C07316=1207.286,250.336,-62.631,-177.060,6.729,148.376
C07317=1207.282,250.584,-62.658,-177.057,6.731,148.376
C07318=1207.277,250.833,-62.684,-177.054,6.733,148.376
C07319=1207.273,251.081,-62.711,-177.052,6.736,148.376
C07320=1207.269,251.330,-62.737,-177.049,6.737,148.375
C07321=1207.264,251.578,-62.764,-177.047,6.740,148.375
C07322=1207.259,251.827,-62.791,-177.044,6.742,148.375
C07323=1207.255,252.075,-62.817,-177.042,6.744,148.375
C07324=1207.251,252.325,-62.844,-177.039,6.746,148.375
C07325=1207.247,252.573,-62.871,-177.037,6.749,148.375
C07326=1207.243,252.821,-62.898,-177.034,6.751,148.374
C07327=1207.238,253.070,-62.925,-177.031,6.753,148.374
C07328=1207.233,253.318,-62.952,-177.029,6.756,148.374
C07329=1207.229,253.566,-62.978,-177.026,6.758,148.374
C07330=1207.224,253.815,-63.005,-177.024,6.760,148.374
C07331=1207.220,254.064,-63.032,-177.021,6.762,148.373
C07332=1207.215,254.312,-63.059,-177.018,6.765,148.373
C07333=1207.211,254.561,-63.085,-177.016,6.767,148.373
C07334=1207.207,254.809,-63.112,-177.014,6.769,148.373
C07335=1207.202,255.058,-63.140,-177.011,6.771,148.372
C07336=1207.197,255.306,-63.167,-177.008,6.774,148.372
C07337=1207.194,255.555,-63.193,-177.006,6.776,148.372
C07338=1207.189,255.804,-63.220,-177.004,6.778,148.372
C07339=1207.185,256.052,-63.248,-177.000,6.781,148.372
C07340=1207.180,256.301,-63.275,-176.998,6.783,148.372
C07341=1207.176,256.549,-63.301,-176.996,6.785,148.371
C07342=1207.171,256.797,-63.328,-176.994,6.787,148.371
C07343=1207.167,257.046,-63.355,-176.990,6.789,148.371
C07344=1207.162,257.294,-63.382,-176.988,6.792,148.371
C07345=1207.157,257.543,-63.409,-176.986,6.793,148.371
C07346=1207.153,257.792,-63.437,-176.983,6.797,148.371
C07347=1207.150,258.039,-63.464,-176.980,6.798,148.370
C07348=1207.145,258.288,-63.491,-176.978,6.801,148.370
C07349=1207.140,258.536,-63.518,-176.975,6.803,148.370
C07350=1207.136,258.785,-63.545,-176.973,6.805,148.370
C07351=1207.131,259.033,-63.572,-176.970,6.807,148.370
C07352=1207.127,259.283,-63.600,-176.968,6.809,148.369
C07353=1207.122,259.531,-63.627,-176.965,6.812,148.369
C07354=1207.118,259.779,-63.654,-176.963,6.814,148.369
C07355=1207.114,260.027,-63.681,-176.960,6.816,148.369
C07356=1207.109,260.276,-63.708,-176.957,6.819,148.369
C07357=1207.105,260.525,-63.735,-176.955,6.821,148.368
C07358=1207.101,260.773,-63.762,-176.953,6.823,148.368
C07359=1207.096,261.021,-63.790,-176.949,6.826,148.368
C07360=1207.092,261.270,-63.817,-176.947,6.828,148.368
C07361=1207.087,261.518,-63.844,-176.945,6.830,148.368
C07362=1207.083,261.767,-63.872,-176.942,6.833,148.368
C07363=1207.079,262.015,-63.900,-176.939,6.835,148.367
C07364=1207.074,262.264,-63.927,-176.937,6.837,148.367
C07365=1207.069,262.512,-63.954,-176.934,6.840,148.367
C07366=1207.065,262.785,-63.984,-176.932,6.842,148.367
C07367=1207.060,263.058,-64.014,-176.929,6.845,148.367
C07368=1207.055,263.331,-64.044,-176.926,6.848,148.367
C07369=1207.050,263.603,-64.074,-176.923,6.850,148.366
C07370=1207.046,263.852,-64.102,-176.921,6.853,148.366
C07371=1207.042,264.100,-64.129,-176.918,6.854,148.366
C07372=1207.037,264.348,-64.156,-176.916,6.857,148.366
C07373=1207.033,264.597,-64.183,-176.913,6.859,148.366
C07374=1207.029,264.846,-64.212,-176.911,6.861,148.366
C07375=1207.024,265.094,-64.239,-176.908,6.863,148.365
C07376=1207.019,265.342,-64.267,-176.905,6.866,148.365
C07377=1207.015,265.591,-64.294,-176.903,6.868,148.365
C07378=1207.011,265.839,-64.322,-176.901,6.870,148.365
C07379=1207.006,266.088,-64.349,-176.898,6.873,148.365
C07380=1207.002,266.336,-64.377,-176.895,6.875,148.365
C07381=1206.998,266.585,-64.404,-176.893,6.877,148.364
C07382=1206.993,266.833,-64.432,-176.890,6.880,148.364
C07383=1206.989,267.081,-64.459,-176.888,6.882,148.364
C07384=1206.985,267.330,-64.487,-176.886,6.885,148.364
C07385=1206.980,267.579,-64.515,-176.883,6.887,148.364
C07386=1206.975,267.826,-64.543,-176.880,6.889,148.364
C07387=1206.971,268.076,-64.570,-176.877,6.892,148.363
C07388=1206.967,268.324,-64.598,-176.875,6.894,148.363
C07389=1206.962,268.571,-64.626,-176.873,6.896,148.363
C07390=1206.958,268.821,-64.653,-176.870,6.899,148.363
C07391=1206.953,269.069,-64.682,-176.868,6.901,148.363
C07392=1206.949,269.317,-64.709,-176.865,6.903,148.363
C07393=1206.945,269.566,-64.737,-176.862,6.906,148.363
C07394=1206.941,269.814,-64.765,-176.860,6.908,148.363
C07395=1206.936,270.063,-64.792,-176.857,6.911,148.362
C07396=1206.931,270.311,-64.820,-176.855,6.913,148.362
C07397=1206.927,270.559,-64.848,-176.852,6.915,148.362
C07398=1206.923,270.808,-64.876,-176.850,6.918,148.362
C07399=1206.919,271.056,-64.903,-176.847,6.920,148.362
C07400=1206.914,271.304,-64.932,-176.845,6.922,148.361
C07401=1206.910,271.553,-64.960,-176.842,6.925,148.361
C07402=1206.905,271.801,-64.987,-176.840,6.927,148.361
C07403=1206.901,272.050,-65.015,-176.837,6.930,148.361
C07404=1206.896,272.298,-65.044,-176.835,6.932,148.361
C07405=1206.893,272.547,-65.072,-176.832,6.934,148.361
C07406=1206.888,272.795,-65.099,-176.829,6.937,148.361
C07407=1206.883,273.043,-65.127,-176.827,6.939,148.361
C07408=1206.879,273.292,-65.155,-176.824,6.942,148.360
C07409=1206.875,273.540,-65.183,-176.822,6.944,148.360
C07410=1206.870,273.789,-65.212,-176.820,6.946,148.360
C07411=1206.866,274.037,-65.240,-176.817,6.949,148.360
C07412=1206.862,274.285,-65.268,-176.814,6.951,148.360
C07413=1206.857,274.533,-65.296,-176.812,6.954,148.360
C07414=1206.853,274.783,-65.323,-176.809,6.956,148.360
C07415=1206.849,275.030,-65.351,-176.806,6.959,148.360
C07416=1206.844,275.279,-65.380,-176.804,6.961,148.359
C07417=1206.840,275.527,-65.408,-176.802,6.963,148.359
C07418=1206.835,275.775,-65.436,-176.799,6.966,148.359
C07419=1206.831,276.024,-65.464,-176.797,6.969,148.359
C07420=1206.827,276.272,-65.492,-176.794,6.971,148.359
C07421=1206.822,276.521,-65.521,-176.792,6.973,148.359
C07422=1206.818,276.769,-65.549,-176.789,6.976,148.359
C07423=1206.813,277.017,-65.577,-176.786,6.978,148.358
C07424=1206.810,277.266,-65.605,-176.784,6.980,148.358
C07425=1206.805,277.514,-65.633,-176.781,6.984,148.358
C07426=1206.801,277.763,-65.662,-176.779,6.985,148.358
C07427=1206.796,278.011,-65.690,-176.776,6.988,148.358
C07428=1206.792,278.260,-65.718,-176.774,6.991,148.358
C07429=1206.787,278.507,-65.746,-176.771,6.994,148.358
C07430=1206.783,278.756,-65.775,-176.769,6.995,148.358
C07431=1206.779,279.004,-65.803,-176.767,6.998,148.357
C07432=1206.774,279.252,-65.832,-176.764,7.001,148.357
C07433=1206.770,279.500,-65.860,-176.761,7.003,148.357
C07434=1206.766,279.749,-65.889,-176.759,7.006,148.357
C07435=1206.762,279.998,-65.917,-176.756,7.008,148.357
C07436=1206.757,280.246,-65.945,-176.754,7.011,148.357
C07437=1206.753,280.495,-65.973,-176.751,7.013,148.357
C07438=1206.748,280.742,-66.002,-176.748,7.016,148.357
C07439=1206.744,280.991,-66.031,-176.746,7.018,148.357
C07440=1206.739,281.239,-66.059,-176.744,7.020,148.356
C07441=1206.735,281.488,-66.088,-176.741,7.023,148.356
C07442=1206.731,281.736,-66.117,-176.739,7.025,148.356
C07443=1206.726,281.984,-66.145,-176.736,7.028,148.356
C07444=1206.723,282.232,-66.173,-176.734,7.030,148.356
C07445=1206.718,282.481,-66.201,-176.731,7.033,148.356
C07446=1206.713,282.729,-66.231,-176.729,7.035,148.356
C07447=1206.710,282.978,-66.259,-176.726,7.038,148.356
C07448=1206.705,283.226,-66.287,-176.723,7.040,148.356
C07449=1206.700,283.475,-66.316,-176.721,7.043,148.355
C07450=1206.697,283.723,-66.345,-176.719,7.045,148.355
C07451=1206.692,283.971,-66.373,-176.716,7.048,148.355
C07452=1206.687,284.220,-66.402,-176.713,7.050,148.355
C07453=1206.684,284.468,-66.431,-176.711,7.052,148.355
C07454=1206.679,284.716,-66.459,-176.708,7.055,148.355
C07455=1206.674,284.964,-66.489,-176.706,7.057,148.355
C07456=1206.671,285.213,-66.517,-176.704,7.060,148.355
C07457=1206.665,285.461,-66.545,-176.701,7.062,148.355
C07458=1206.661,285.709,-66.575,-176.698,7.065,148.355
C07459=1206.658,285.958,-66.603,-176.696,7.068,148.355
C07460=1206.653,286.205,-66.632,-176.694,7.071,148.354
C07461=1206.648,286.454,-66.661,-176.691,7.072,148.354
C07462=1206.644,286.702,-66.690,-176.688,7.076,148.354
C07463=1206.640,286.950,-66.718,-176.686,7.078,148.354
C07464=1206.636,287.199,-66.747,-176.683,7.081,148.354
C07465=1206.631,287.447,-66.776,-176.681,7.083,148.354
C07466=1206.626,287.695,-66.805,-176.678,7.086,148.354
C07467=1206.623,287.944,-66.833,-176.676,7.088,148.354
C07468=1206.618,288.192,-66.863,-176.673,7.091,148.354
C07469=1206.614,288.441,-66.892,-176.671,7.093,148.354
C07470=1206.609,288.714,-66.924,-176.668,7.096,148.354
C07471=1206.605,288.989,-66.956,-176.665,7.099,148.353
C07472=1206.599,289.263,-66.988,-176.663,7.102,148.353
C07473=1206.595,289.537,-67.020,-176.660,7.105,148.353
C07474=1206.590,289.786,-67.049,-176.658,7.107,148.353
C07475=1206.586,290.033,-67.077,-176.655,7.110,148.353
C07476=1206.582,290.282,-67.106,-176.653,7.112,148.353
C07477=1206.577,290.531,-67.136,-176.650,7.115,148.353
C07478=1206.573,290.779,-67.165,-176.648,7.117,148.353
C07479=1206.569,291.028,-67.194,-176.645,7.120,148.353
C07480=1206.564,291.275,-67.223,-176.643,7.122,148.353
C07481=1206.560,291.523,-67.252,-176.640,7.125,148.353
C07482=1206.556,291.772,-67.282,-176.638,7.127,148.352
C07483=1206.552,292.020,-67.310,-176.635,7.130,148.352
C07484=1206.548,292.269,-67.339,-176.633,7.132,148.352
C07485=1206.543,292.516,-67.369,-176.630,7.135,148.352
C07486=1206.539,292.764,-67.398,-176.628,7.138,148.352
C07487=1206.534,293.013,-67.427,-176.625,7.141,148.352
C07488=1206.530,293.262,-67.456,-176.623,7.143,148.352
C07489=1206.526,293.510,-67.486,-176.620,7.146,148.352
C07490=1206.521,293.757,-67.515,-176.618,7.148,148.352
C07491=1206.517,294.006,-67.544,-176.615,7.151,148.352
C07492=1206.513,294.254,-67.574,-176.612,7.154,148.352
C07493=1206.508,294.503,-67.602,-176.610,7.156,148.352
C07494=1206.504,294.751,-67.632,-176.608,7.159,148.352
C07495=1206.500,294.999,-67.661,-176.605,7.161,148.352
C07496=1206.496,295.248,-67.691,-176.603,7.164,148.352
C07497=1206.491,295.495,-67.720,-176.601,7.166,148.352
C07498=1206.487,295.743,-67.749,-176.598,7.169,148.352
C07499=1206.482,295.992,-67.779,-176.595,7.171,148.351
C07500=1206.478,296.240,-67.808,-176.593,7.174,148.351
C07501=1206.474,296.488,-67.838,-176.591,7.177,148.351
C07502=1206.470,296.737,-67.867,-176.588,7.180,148.351
C07503=1206.466,296.985,-67.897,-176.586,7.182,148.351
C07504=1206.462,297.233,-67.926,-176.583,7.185,148.351
C07505=1206.457,297.481,-67.955,-176.580,7.188,148.351
C07506=1206.453,297.729,-67.984,-176.578,7.190,148.351
C07507=1206.448,297.978,-68.015,-176.576,7.193,148.351
C07508=1206.443,298.226,-68.044,-176.573,7.195,148.351
C07509=1206.439,298.474,-68.073,-176.571,7.198,148.351
C07510=1206.435,298.722,-68.103,-176.569,7.201,148.351
C07511=1206.431,298.971,-68.132,-176.566,7.204,148.351
C07512=1206.427,299.219,-68.162,-176.564,7.206,148.351
C07513=1206.423,299.467,-68.191,-176.561,7.209,148.351
C07514=1206.418,299.715,-68.221,-176.559,7.211,148.351
C07515=1206.413,299.964,-68.251,-176.556,7.214,148.351
C07516=1206.409,300.212,-68.280,-176.554,7.217,148.351
C07517=1206.405,300.460,-68.310,-176.551,7.219,148.351
C07518=1206.401,300.708,-68.340,-176.549,7.222,148.351
C07519=1206.397,300.956,-68.369,-176.547,7.224,148.351
C07520=1206.392,301.205,-68.399,-176.544,7.227,148.351
C07521=1206.388,301.453,-68.429,-176.542,7.230,148.351
C07522=1206.384,301.701,-68.459,-176.539,7.233,148.350
C07523=1206.380,301.949,-68.488,-176.536,7.236,148.350
C07524=1206.376,302.197,-68.518,-176.534,7.238,148.350
C07525=1206.371,302.446,-68.548,-176.532,7.241,148.350
C07526=1206.367,302.694,-68.578,-176.530,7.243,148.350
C07527=1206.363,302.942,-68.608,-176.527,7.246,148.350
C07528=1206.359,303.190,-68.637,-176.525,7.248,148.350
C07529=1206.354,303.439,-68.667,-176.522,7.251,148.350
C07530=1206.350,303.686,-68.697,-176.519,7.254,148.350
C07531=1206.346,303.935,-68.727,-176.517,7.257,148.350
C07532=1206.341,304.183,-68.757,-176.515,7.260,148.350
C07533=1206.337,304.431,-68.787,-176.512,7.262,148.350
C07534=1206.333,304.679,-68.816,-176.510,7.265,148.350
C07535=1206.328,304.928,-68.846,-176.508,7.267,148.350
C07536=1206.324,305.175,-68.877,-176.505,7.270,148.350
C07537=1206.320,305.424,-68.906,-176.502,7.273,148.350
C07538=1206.315,305.672,-68.937,-176.500,7.275,148.350
C07539=1206.311,305.920,-68.966,-176.497,7.278,148.350
C07540=1206.307,306.168,-68.996,-176.495,7.281,148.350
C07541=1206.302,306.416,-69.026,-176.493,7.284,148.350
C07542=1206.298,306.664,-69.056,-176.490,7.286,148.350
C07543=1206.294,306.912,-69.086,-176.488,7.289,148.350
C07544=1206.289,307.161,-69.116,-176.485,7.292,148.350
C07545=1206.285,307.408,-69.146,-176.483,7.294,148.350
C07546=1206.280,307.657,-69.176,-176.481,7.297,148.350
C07547=1206.277,307.905,-69.207,-176.479,7.300,148.350
C07548=1206.272,308.154,-69.237,-176.476,7.303,148.350
C07549=1206.268,308.401,-69.267,-176.473,7.306,148.350
C07550=1206.264,308.650,-69.297,-176.471,7.308,148.350
C07551=1206.259,308.898,-69.327,-176.468,7.311,148.350
C07552=1206.256,309.145,-69.357,-176.466,7.313,148.350
C07553=1206.251,309.394,-69.388,-176.464,7.316,148.350
C07554=1206.247,309.642,-69.418,-176.461,7.319,148.350
C07555=1206.242,309.890,-69.448,-176.459,7.322,148.350
C07556=1206.239,310.138,-69.478,-176.457,7.325,148.350
C07557=1206.234,310.386,-69.509,-176.454,7.327,148.350
C07558=1206.230,310.635,-69.538,-176.452,7.330,148.350
C07559=1206.225,310.883,-69.569,-176.449,7.333,148.350
C07560=1206.221,311.130,-69.599,-176.447,7.335,148.350
C07561=1206.216,311.379,-69.629,-176.445,7.338,148.350
C07562=1206.213,311.627,-69.660,-176.443,7.341,148.350
C07563=1206.208,311.875,-69.691,-176.440,7.344,148.350
C07564=1206.204,312.123,-69.720,-176.437,7.347,148.350
C07565=1206.200,312.371,-69.751,-176.435,7.349,148.350
C07566=1206.195,312.619,-69.782,-176.432,7.352,148.350
C07567=1206.191,312.867,-69.812,-176.431,7.354,148.350
C07568=1206.187,313.116,-69.842,-176.428,7.357,148.350
C07569=1206.183,313.364,-69.873,-176.425,7.360,148.350
C07570=1206.178,313.612,-69.903,-176.423,7.363,148.350
C07571=1206.174,313.860,-69.933,-176.421,7.366,148.350
C07572=1206.170,314.107,-69.964,-176.419,7.368,148.350
C07573=1206.166,314.357,-69.995,-176.416,7.371,148.350
C07574=1206.161,314.633,-70.029,-176.414,7.374,148.350
C07575=1206.157,314.908,-70.063,-176.411,7.377,148.350
C07576=1206.152,315.184,-70.096,-176.408,7.380,148.350
C07577=1206.147,315.460,-70.130,-176.406,7.383,148.350
C07578=1206.143,315.709,-70.162,-176.403,7.387,148.350
C07579=1206.138,315.957,-70.192,-176.401,7.389,148.350
C07580=1206.134,316.204,-70.222,-176.399,7.392,148.350
C07581=1206.129,316.453,-70.253,-176.396,7.395,148.350
C07582=1206.125,316.702,-70.284,-176.394,7.397,148.350
C07583=1206.122,316.949,-70.314,-176.392,7.401,148.350
C07584=1206.117,317.197,-70.345,-176.389,7.403,148.350
C07585=1206.113,317.446,-70.376,-176.387,7.406,148.350
C07586=1206.108,317.694,-70.406,-176.385,7.409,148.351
C07587=1206.104,317.942,-70.437,-176.382,7.411,148.350
C07588=1206.100,318.190,-70.467,-176.380,7.414,148.350
C07589=1206.096,318.438,-70.499,-176.377,7.418,148.351
C07590=1206.092,318.686,-70.529,-176.375,7.420,148.351
C07591=1206.088,318.933,-70.560,-176.373,7.423,148.351
C07592=1206.084,319.182,-70.591,-176.371,7.425,148.351
C07593=1206.079,319.430,-70.622,-176.368,7.428,148.351
C07594=1206.074,319.678,-70.653,-176.366,7.431,148.351
C07595=1206.071,319.926,-70.683,-176.364,7.434,148.351
C07596=1206.067,320.174,-70.714,-176.361,7.437,148.351
C07597=1206.062,320.422,-70.745,-176.359,7.440,148.351
C07598=1206.058,320.671,-70.776,-176.357,7.442,148.351
C07599=1206.053,320.919,-70.807,-176.354,7.446,148.351
C07600=1206.050,321.166,-70.838,-176.352,7.448,148.351
C07601=1206.046,321.414,-70.869,-176.349,7.451,148.351
C07602=1206.041,321.662,-70.900,-176.347,7.454,148.351
C07603=1206.036,321.910,-70.930,-176.345,7.456,148.351
C07604=1206.032,322.159,-70.961,-176.342,7.459,148.351
C07605=1206.028,322.406,-70.993,-176.340,7.463,148.351
C07606=1206.025,322.655,-71.023,-176.338,7.465,148.351
C07607=1206.020,322.903,-71.054,-176.336,7.468,148.352
C07608=1206.016,323.151,-71.085,-176.334,7.470,148.352
C07609=1206.012,323.399,-71.117,-176.331,7.474,148.352
C07610=1206.007,323.647,-71.148,-176.329,7.477,148.352
C07611=1206.003,323.895,-71.179,-176.327,7.479,148.352
C07612=1205.999,324.143,-71.210,-176.325,7.482,148.352
C07613=1205.994,324.390,-71.241,-176.322,7.485,148.352
C07614=1205.990,324.639,-71.272,-176.320,7.488,148.352
C07615=1205.986,324.886,-71.304,-176.318,7.491,148.352
C07616=1205.982,325.135,-71.335,-176.315,7.493,148.352
C07617=1205.977,325.383,-71.366,-176.313,7.497,148.352
C07618=1205.974,325.631,-71.397,-176.311,7.500,148.352
C07619=1205.970,325.879,-71.428,-176.309,7.502,148.352
C07620=1205.966,326.126,-71.459,-176.306,7.505,148.352
C07621=1205.962,326.375,-71.490,-176.304,7.508,148.352
C07622=1205.957,326.623,-71.521,-176.302,7.511,148.353
C07623=1205.953,326.871,-71.553,-176.299,7.514,148.353
C07624=1205.949,327.119,-71.584,-176.298,7.516,148.353
C07625=1205.944,327.367,-71.616,-176.295,7.519,148.353
C07626=1205.940,327.615,-71.647,-176.293,7.523,148.353
C07627=1205.936,327.863,-71.679,-176.290,7.525,148.353
C07628=1205.931,328.111,-71.709,-176.288,7.528,148.353
C07629=1205.928,328.359,-71.741,-176.286,7.531,148.353
C07630=1205.923,328.607,-71.772,-176.284,7.534,148.353
C07631=1205.919,328.855,-71.804,-176.281,7.537,148.353
C07632=1205.915,329.103,-71.835,-176.279,7.540,148.354
C07633=1205.911,329.351,-71.866,-176.277,7.542,148.354
C07634=1205.907,329.598,-71.898,-176.275,7.546,148.354
C07635=1205.903,329.847,-71.929,-176.273,7.548,148.354
C07636=1205.898,330.094,-71.960,-176.270,7.551,148.354
C07637=1205.894,330.343,-71.992,-176.268,7.554,148.354
C07638=1205.889,330.591,-72.024,-176.266,7.557,148.354
C07639=1205.885,330.839,-72.056,-176.264,7.560,148.354
C07640=1205.881,331.087,-72.086,-176.261,7.563,148.354
C07641=1205.877,331.335,-72.118,-176.259,7.566,148.354
C07642=1205.873,331.582,-72.150,-176.257,7.569,148.354
C07643=1205.869,331.831,-72.181,-176.255,7.571,148.355
C07644=1205.865,332.078,-72.212,-176.253,7.574,148.355
C07645=1205.860,332.326,-72.245,-176.250,7.577,148.355
C07646=1205.856,332.575,-72.276,-176.249,7.580,148.355
C07647=1205.852,332.822,-72.307,-176.246,7.583,148.355
C07648=1205.848,333.070,-72.339,-176.244,7.586,148.355
C07649=1205.844,333.318,-72.371,-176.242,7.589,148.355
C07650=1205.839,333.566,-72.403,-176.239,7.592,148.355
C07651=1205.835,333.814,-72.434,-176.237,7.595,148.356
C07652=1205.831,334.062,-72.466,-176.235,7.598,148.356
C07653=1205.827,334.310,-72.497,-176.233,7.601,148.356
C07654=1205.822,334.558,-72.530,-176.231,7.603,148.356
C07655=1205.819,334.806,-72.561,-176.229,7.607,148.356
C07656=1205.814,335.054,-72.592,-176.226,7.610,148.356
C07657=1205.810,335.302,-72.624,-176.225,7.612,148.356
C07658=1205.806,335.550,-72.656,-176.222,7.616,148.357
C07659=1205.801,335.798,-72.688,-176.220,7.619,148.357
C07660=1205.798,336.046,-72.720,-176.218,7.621,148.357
C07661=1205.793,336.294,-72.752,-176.216,7.624,148.357
C07662=1205.789,336.541,-72.784,-176.214,7.627,148.357
C07663=1205.785,336.789,-72.816,-176.212,7.630,148.357
C07664=1205.780,337.037,-72.848,-176.209,7.633,148.357
C07665=1205.777,337.285,-72.879,-176.207,7.636,148.357
C07666=1205.773,337.534,-72.911,-176.205,7.639,148.358
C07667=1205.768,337.781,-72.943,-176.203,7.642,148.358
C07668=1205.764,338.029,-72.975,-176.201,7.645,148.358
C07669=1205.760,338.277,-73.006,-176.198,7.648,148.358
C07670=1205.755,338.525,-73.038,-176.197,7.650,148.358
C07671=1205.751,338.773,-73.070,-176.195,7.654,148.358
C07672=1205.748,339.020,-73.103,-176.192,7.657,148.359
C07673=1205.743,339.269,-73.135,-176.191,7.659,148.359
C07674=1205.739,339.516,-73.167,-176.188,7.662,148.359
C07675=1205.735,339.765,-73.199,-176.186,7.666,148.359
C07676=1205.731,340.013,-73.231,-176.184,7.668,148.359
C07677=1205.727,340.260,-73.263,-176.182,7.672,148.359
C07678=1205.722,340.538,-73.299,-176.180,7.675,148.360
C07679=1205.717,340.817,-73.335,-176.177,7.678,148.360
C07680=1205.712,341.095,-73.371,-176.175,7.681,148.360
C07681=1205.708,341.373,-73.407,-176.173,7.685,148.360
C07682=1205.704,341.621,-73.439,-176.170,7.688,148.360
C07683=1205.699,341.869,-73.471,-176.169,7.691,148.361
C07684=1205.695,342.117,-73.503,-176.166,7.694,148.361
C07685=1205.691,342.365,-73.535,-176.164,7.697,148.361
C07686=1205.687,342.613,-73.568,-176.162,7.699,148.361
C07687=1205.683,342.860,-73.600,-176.160,7.703,148.361
C07688=1205.678,343.109,-73.632,-176.158,7.705,148.361
C07689=1205.675,343.357,-73.664,-176.156,7.709,148.362
C07690=1205.670,343.604,-73.697,-176.154,7.712,148.362
C07691=1205.666,343.852,-73.729,-176.152,7.715,148.362
C07692=1205.662,344.100,-73.761,-176.150,7.718,148.362
C07693=1205.658,344.348,-73.793,-176.148,7.720,148.362
C07694=1205.654,344.596,-73.826,-176.146,7.724,148.363
C07695=1205.649,344.843,-73.858,-176.144,7.727,148.363
C07696=1205.645,345.091,-73.890,-176.142,7.730,148.363
C07697=1205.641,345.339,-73.923,-176.140,7.733,148.363
C07698=1205.637,345.587,-73.955,-176.137,7.736,148.363
C07699=1205.633,345.836,-73.987,-176.136,7.738,148.363
C07700=1205.628,346.083,-74.020,-176.133,7.742,148.364
C07701=1205.624,346.331,-74.052,-176.132,7.744,148.364
C07702=1205.620,346.578,-74.085,-176.130,7.748,148.364
C07703=1205.617,346.826,-74.117,-176.127,7.751,148.364
C07704=1205.612,347.075,-74.149,-176.126,7.754,148.364
C07705=1205.608,347.322,-74.183,-176.124,7.757,148.365
C07706=1205.604,347.570,-74.214,-176.122,7.760,148.365
C07707=1205.600,347.818,-74.247,-176.120,7.763,148.365
C07708=1205.595,348.066,-74.280,-176.118,7.766,148.365
C07709=1205.592,348.313,-74.312,-176.116,7.769,148.366
C07710=1205.587,348.562,-74.345,-176.114,7.772,148.366
C07711=1205.583,348.809,-74.378,-176.112,7.775,148.366
C07712=1205.579,349.057,-74.409,-176.110,7.778,148.366
C07713=1205.575,349.304,-74.442,-176.108,7.781,148.367
C07714=1205.570,349.553,-74.475,-176.106,7.784,148.367
C07715=1205.567,349.800,-74.507,-176.104,7.787,148.367
C07716=1205.562,350.049,-74.540,-176.102,7.790,148.367
C07717=1205.558,350.296,-74.573,-176.100,7.793,148.367
C07718=1205.554,350.545,-74.605,-176.098,7.797,148.368
C07719=1205.550,350.791,-74.638,-176.097,7.799,148.368
C07720=1205.545,351.040,-74.670,-176.095,7.803,148.368
C07721=1205.541,351.287,-74.703,-176.093,7.805,148.368
C07722=1205.537,351.535,-74.736,-176.091,7.808,148.369
C07723=1205.533,351.783,-74.768,-176.089,7.811,148.369
C07724=1205.529,352.031,-74.801,-176.087,7.815,148.369
C07725=1205.525,352.279,-74.835,-176.085,7.818,148.369
C07726=1205.521,352.527,-74.867,-176.083,7.820,148.370
C07727=1205.517,352.775,-74.900,-176.081,7.824,148.370
C07728=1205.513,353.022,-74.933,-176.079,7.826,148.370
C07729=1205.509,353.271,-74.965,-176.078,7.830,148.370
C07730=1205.505,353.518,-74.998,-176.076,7.832,148.371
C07731=1205.500,353.765,-75.031,-176.074,7.836,148.371
C07732=1205.496,354.013,-75.064,-176.072,7.839,148.371
C07733=1205.492,354.261,-75.096,-176.070,7.842,148.371
C07734=1205.488,354.509,-75.129,-176.068,7.845,148.372
C07735=1205.484,354.756,-75.162,-176.067,7.848,148.372
C07736=1205.480,355.004,-75.196,-176.064,7.851,148.372
C07737=1205.475,355.253,-75.228,-176.063,7.854,148.372
C07738=1205.471,355.500,-75.261,-176.061,7.857,148.373
C07739=1205.467,355.748,-75.294,-176.059,7.861,148.373
C07740=1205.463,355.995,-75.327,-176.057,7.863,148.373
C07741=1205.459,356.243,-75.360,-176.055,7.867,148.374
C07742=1205.455,356.492,-75.392,-176.054,7.869,148.374
C07743=1205.451,356.739,-75.426,-176.052,7.873,148.374
C07744=1205.447,356.987,-75.459,-176.050,7.875,148.374
C07745=1205.442,357.235,-75.492,-176.048,7.879,148.375
C07746=1205.438,357.482,-75.525,-176.046,7.882,148.375
C07747=1205.434,357.730,-75.558,-176.045,7.885,148.375
C07748=1205.430,357.978,-75.591,-176.043,7.889,148.376
C07749=1205.426,358.226,-75.625,-176.041,7.891,148.376
C07750=1205.422,358.473,-75.658,-176.039,7.894,148.376
C07751=1205.418,358.721,-75.691,-176.038,7.897,148.376
C07752=1205.413,358.969,-75.724,-176.035,7.901,148.377
C07753=1205.409,359.217,-75.757,-176.034,7.903,148.377
C07754=1205.405,359.464,-75.790,-176.032,7.907,148.377
C07755=1205.401,359.712,-75.824,-176.031,7.910,148.378
C07756=1205.397,359.960,-75.857,-176.029,7.913,148.378
C07757=1205.393,360.207,-75.890,-176.027,7.916,148.378
C07758=1205.389,360.455,-75.923,-176.025,7.919,148.379
C07759=1205.385,360.704,-75.956,-176.024,7.922,148.379
C07760=1205.381,360.951,-75.990,-176.022,7.925,148.379
C07761=1205.377,361.199,-76.023,-176.021,7.928,148.380
C07762=1205.373,361.447,-76.056,-176.018,7.931,148.380
C07763=1205.369,361.695,-76.089,-176.017,7.934,148.380
C07764=1205.364,361.942,-76.122,-176.015,7.938,148.380
C07765=1205.360,362.190,-76.155,-176.014,7.940,148.381
C07766=1205.356,362.438,-76.189,-176.012,7.944,148.381
C07767=1205.352,362.685,-76.222,-176.010,7.947,148.381
C07768=1205.348,362.933,-76.255,-176.009,7.950,148.382
C07769=1205.344,363.180,-76.289,-176.007,7.953,148.382
C07770=1205.340,363.428,-76.322,-176.005,7.956,148.382
C07771=1205.336,363.676,-76.355,-176.004,7.959,148.383
C07772=1205.332,363.924,-76.389,-176.002,7.962,148.383
C07773=1205.328,364.172,-76.422,-176.001,7.965,148.383
C07774=1205.324,364.420,-76.455,-175.999,7.969,148.384
C07775=1205.319,364.667,-76.489,-175.997,7.971,148.384
C07776=1205.315,364.915,-76.523,-175.996,7.974,148.384
C07777=1205.311,365.163,-76.556,-175.994,7.978,148.385
C07778=1205.307,365.410,-76.589,-175.993,7.981,148.385
C07779=1205.304,365.658,-76.623,-175.991,7.984,148.386
C07780=1205.300,365.906,-76.656,-175.989,7.987,148.386
C07781=1205.295,366.154,-76.689,-175.988,7.990,148.386
C07782=1205.291,366.434,-76.728,-175.987,7.993,148.387
C07783=1205.285,366.714,-76.766,-175.985,7.997,148.387
C07784=1205.281,366.995,-76.803,-175.983,8.001,148.388
C07785=1205.276,367.276,-76.842,-175.981,8.004,148.388
C07786=1205.272,367.523,-76.875,-175.980,8.007,148.388
C07787=1205.268,367.770,-76.909,-175.978,8.010,148.389
C07788=1205.265,368.019,-76.942,-175.977,8.013,148.389
C07789=1205.261,368.267,-76.975,-175.975,8.016,148.390
C07790=1205.256,368.514,-77.010,-175.974,8.020,148.390
C07791=1205.252,368.762,-77.043,-175.972,8.022,148.390
C07792=1205.248,369.009,-77.077,-175.971,8.025,148.391
C07793=1205.244,369.257,-77.110,-175.969,8.029,148.391
C07794=1205.240,369.505,-77.144,-175.968,8.031,148.391
C07795=1205.236,369.752,-77.178,-175.967,8.034,148.392
C07796=1205.232,370.000,-77.211,-175.965,8.038,148.392
C07797=1205.228,370.247,-77.245,-175.964,8.041,148.393
C07798=1205.223,370.495,-77.279,-175.962,8.043,148.393
C07799=1205.220,370.743,-77.313,-175.961,8.047,148.393
C07800=1205.216,370.991,-77.346,-175.959,8.050,148.394
C07801=1205.211,371.238,-77.381,-175.958,8.053,148.394
C07802=1205.207,371.486,-77.414,-175.957,8.056,148.395
C07803=1205.204,371.734,-77.448,-175.955,8.059,148.395
C07804=1205.199,371.982,-77.482,-175.954,8.062,148.395
C07805=1205.195,372.229,-77.516,-175.953,8.065,148.396
C07806=1205.191,372.477,-77.549,-175.952,8.068,148.396
C07807=1205.186,372.724,-77.583,-175.950,8.071,148.397
C07808=1205.183,372.972,-77.617,-175.949,8.074,148.397
C07809=1205.179,373.220,-77.651,-175.947,8.077,148.397
C07810=1205.174,373.468,-77.684,-175.947,8.080,148.398
C07811=1205.170,373.715,-77.718,-175.945,8.084,148.398
C07812=1205.167,373.963,-77.752,-175.944,8.086,148.399
C07813=1205.162,374.211,-77.786,-175.942,8.089,148.399
C07814=1205.158,374.458,-77.820,-175.941,8.092,148.400
C07815=1205.155,374.706,-77.854,-175.940,8.095,148.400
C07816=1205.150,374.954,-77.888,-175.939,8.098,148.400
C07817=1205.146,375.201,-77.921,-175.937,8.101,148.401
C07818=1205.141,375.449,-77.956,-175.936,8.104,148.401
C07819=1205.138,375.697,-77.990,-175.935,8.107,148.402
C07820=1205.134,375.944,-78.023,-175.934,8.110,148.402
C07821=1205.130,376.192,-78.058,-175.933,8.113,148.403
C07822=1205.126,376.439,-78.092,-175.932,8.116,148.403
C07823=1205.121,376.688,-78.126,-175.931,8.119,148.404
C07824=1205.118,376.935,-78.160,-175.929,8.122,148.404
C07825=1205.114,377.182,-78.193,-175.928,8.125,148.404
C07826=1205.110,377.430,-78.227,-175.927,8.128,148.405
C07827=1205.106,377.678,-78.261,-175.926,8.131,148.405
C07828=1205.101,377.925,-78.296,-175.925,8.134,148.406
C07829=1205.098,378.173,-78.330,-175.923,8.137,148.406
C07830=1205.093,378.421,-78.364,-175.923,8.140,148.407
C07831=1205.089,378.668,-78.398,-175.921,8.143,148.407
C07832=1205.085,378.916,-78.433,-175.920,8.145,148.408
C07833=1205.081,379.163,-78.466,-175.919,8.149,148.408
C07834=1205.076,379.411,-78.500,-175.918,8.151,148.409
C07835=1205.073,379.659,-78.534,-175.917,8.154,148.409
C07836=1205.069,379.906,-78.569,-175.916,8.157,148.410
C07837=1205.065,380.154,-78.603,-175.915,8.160,148.410
C07838=1205.061,380.402,-78.638,-175.914,8.163,148.410
C07839=1205.057,380.649,-78.671,-175.913,8.166,148.411
C07840=1205.052,380.897,-78.705,-175.912,8.169,148.411
C07841=1205.049,381.145,-78.739,-175.911,8.172,148.412
C07842=1205.044,381.392,-78.774,-175.910,8.175,148.412
C07843=1205.041,381.639,-78.808,-175.909,8.178,148.413
C07844=1205.037,381.887,-78.843,-175.908,8.181,148.413
C07845=1205.033,382.134,-78.876,-175.907,8.183,148.414
C07846=1205.028,382.382,-78.910,-175.906,8.187,148.414
C07847=1205.025,382.630,-78.944,-175.905,8.189,148.415
C07848=1205.020,382.878,-78.979,-175.904,8.192,148.415
C07849=1205.016,383.126,-79.014,-175.903,8.195,148.416
C07850=1205.012,383.373,-79.048,-175.902,8.198,148.416
C07851=1205.008,383.620,-79.082,-175.901,8.200,148.417
C07852=1205.004,383.868,-79.116,-175.901,8.203,148.417
C07853=1205.000,384.116,-79.151,-175.899,8.206,148.418
C07854=1204.996,384.364,-79.186,-175.899,8.209,148.418
C07855=1204.992,384.611,-79.219,-175.897,8.212,148.419
C07856=1204.988,384.858,-79.254,-175.897,8.215,148.419
C07857=1204.984,385.106,-79.288,-175.896,8.218,148.420
C07858=1204.980,385.353,-79.323,-175.895,8.220,148.420
C07859=1204.976,385.602,-79.357,-175.894,8.223,148.421
C07860=1204.972,385.849,-79.391,-175.893,8.226,148.421
C07861=1204.967,386.096,-79.426,-175.892,8.229,148.422
C07862=1204.964,386.344,-79.460,-175.892,8.231,148.422
C07863=1204.960,386.591,-79.495,-175.891,8.234,148.423
C07864=1204.956,386.839,-79.529,-175.890,8.238,148.423
C07865=1204.952,387.087,-79.563,-175.889,8.240,148.424
C07866=1204.947,387.334,-79.598,-175.889,8.243,148.424
C07867=1204.943,387.582,-79.633,-175.888,8.245,148.424
C07868=1204.939,387.829,-79.666,-175.887,8.249,148.425
C07869=1204.935,388.077,-79.701,-175.886,8.252,148.426
C07870=1204.931,388.325,-79.736,-175.885,8.254,148.426
C07871=1204.928,388.573,-79.770,-175.885,8.257,148.427
C07872=1204.923,388.820,-79.804,-175.884,8.260,148.427
C07873=1204.919,389.068,-79.839,-175.883,8.262,148.427
C07874=1204.915,389.315,-79.873,-175.882,8.265,148.428
C07875=1204.911,389.562,-79.908,-175.882,8.268,148.429
C07876=1204.907,389.810,-79.943,-175.881,8.270,148.429
C07877=1204.903,390.057,-79.977,-175.880,8.273,148.430
C07878=1204.899,390.305,-80.012,-175.879,8.276,148.430
C07879=1204.895,390.553,-80.046,-175.879,8.278,148.431
C07880=1204.891,390.801,-80.081,-175.878,8.281,148.431
C07881=1204.887,391.048,-80.115,-175.878,8.284,148.432
C07882=1204.883,391.296,-80.150,-175.877,8.287,148.432
C07883=1204.879,391.543,-80.185,-175.876,8.289,148.433
C07884=1204.875,391.791,-80.219,-175.876,8.292,148.433
C07885=1204.871,392.038,-80.254,-175.875,8.295,148.434
C07886=1204.867,392.320,-80.294,-175.874,8.298,148.434
C07887=1204.862,392.603,-80.333,-175.874,8.300,148.435
C07888=1204.857,392.886,-80.373,-175.873,8.303,148.435
C07889=1204.852,393.169,-80.412,-175.872,8.306,148.436
C07890=1204.849,393.416,-80.446,-175.871,8.309,148.436
C07891=1204.845,393.664,-80.482,-175.871,8.312,148.437
C07892=1204.840,393.911,-80.516,-175.870,8.315,148.438
C07893=1204.836,394.159,-80.551,-175.870,8.317,148.438
C07894=1204.832,394.406,-80.585,-175.869,8.320,148.439
C07895=1204.829,394.654,-80.620,-175.868,8.322,148.439
C07896=1204.824,394.901,-80.655,-175.868,8.325,148.440
C07897=1204.820,395.149,-80.690,-175.867,8.327,148.440
C07898=1204.816,395.397,-80.724,-175.866,8.330,148.441
C07899=1204.813,395.644,-80.759,-175.866,8.332,148.441
C07900=1204.808,395.891,-80.793,-175.866,8.335,148.442
C07901=1204.804,396.140,-80.828,-175.865,8.338,148.442
C07902=1204.800,396.387,-80.863,-175.864,8.340,148.443
C07903=1204.796,396.634,-80.898,-175.864,8.343,148.443
C07904=1204.792,396.882,-80.932,-175.863,8.345,148.444
C07905=1204.788,397.130,-80.967,-175.863,8.347,148.444
C07906=1204.784,397.376,-81.002,-175.862,8.351,148.445
C07907=1204.780,397.625,-81.037,-175.862,8.352,148.445
C07908=1204.775,397.872,-81.072,-175.861,8.356,148.446
C07909=1204.772,398.120,-81.107,-175.861,8.358,148.446
C07910=1204.768,398.367,-81.141,-175.861,8.360,148.447
C07911=1204.764,398.615,-81.176,-175.860,8.363,148.447
C07912=1204.760,398.862,-81.211,-175.859,8.365,148.448
C07913=1204.756,399.110,-81.246,-175.859,8.367,148.448
C07914=1204.752,399.358,-81.281,-175.858,8.371,148.449
C07915=1204.747,399.605,-81.316,-175.858,8.373,148.449
C07916=1204.743,399.853,-81.351,-175.858,8.375,148.450
C07917=1204.740,400.099,-81.385,-175.857,8.377,148.450
C07918=1204.736,400.347,-81.420,-175.856,8.380,148.451
C07919=1204.731,400.595,-81.455,-175.856,8.382,148.451
C07920=1204.728,400.842,-81.490,-175.856,8.385,148.452
C07921=1204.723,401.090,-81.525,-175.855,8.388,148.453
C07922=1204.720,401.337,-81.560,-175.854,8.390,148.453
C07923=1204.716,401.585,-81.595,-175.854,8.392,148.453
C07924=1204.711,401.833,-81.629,-175.854,8.394,148.454
C07925=1204.707,402.080,-81.665,-175.853,8.397,148.455
C07926=1204.704,402.327,-81.699,-175.853,8.400,148.455
C07927=1204.700,402.575,-81.734,-175.852,8.402,148.455
C07928=1204.695,402.822,-81.769,-175.852,8.404,148.456
C07929=1204.692,403.070,-81.804,-175.852,8.406,148.456
C07930=1204.688,403.318,-81.839,-175.851,8.409,148.457
C07931=1204.683,403.565,-81.874,-175.851,8.412,148.458
C07932=1204.679,403.813,-81.909,-175.850,8.414,148.458
C07933=1204.675,404.060,-81.944,-175.850,8.416,148.458
C07934=1204.671,404.308,-81.979,-175.850,8.418,148.459
C07935=1204.668,404.555,-82.015,-175.850,8.420,148.459
C07936=1204.663,404.803,-82.049,-175.849,8.423,148.460
C07937=1204.659,405.050,-82.085,-175.849,8.426,148.461
C07938=1204.655,405.297,-82.119,-175.848,8.428,148.461
C07939=1204.652,405.545,-82.154,-175.848,8.430,148.461
C07940=1204.648,405.793,-82.189,-175.847,8.432,148.462
C07941=1204.644,406.040,-82.224,-175.847,8.435,148.463
C07942=1204.640,406.288,-82.259,-175.847,8.437,148.463
C07943=1204.635,406.535,-82.294,-175.846,8.440,148.463
C07944=1204.631,406.783,-82.329,-175.846,8.442,148.464
C07945=1204.628,407.030,-82.365,-175.845,8.444,148.465
C07946=1204.623,407.278,-82.399,-175.845,8.446,148.465
C07947=1204.619,407.525,-82.435,-175.845,8.449,148.466
C07948=1204.615,407.773,-82.469,-175.844,8.451,148.466
C07949=1204.611,408.020,-82.505,-175.844,8.453,148.466
C07950=1204.608,408.268,-82.540,-175.844,8.455,148.467
C07951=1204.603,408.515,-82.575,-175.844,8.457,148.468
C07952=1204.599,408.762,-82.610,-175.843,8.459,148.468
C07953=1204.595,409.011,-82.645,-175.843,8.462,148.468
C07954=1204.591,409.257,-82.680,-175.842,8.464,148.469
C07955=1204.587,409.505,-82.715,-175.842,8.466,148.469
C07956=1204.583,409.752,-82.750,-175.842,8.468,148.470
C07957=1204.579,410.000,-82.786,-175.841,8.470,148.470
C07958=1204.575,410.248,-82.821,-175.841,8.473,148.471
C07959=1204.571,410.495,-82.856,-175.841,8.475,148.471
C07960=1204.567,410.742,-82.891,-175.841,8.477,148.472
C07961=1204.563,410.990,-82.926,-175.840,8.479,148.472
C07962=1204.559,411.237,-82.961,-175.840,8.481,148.473
C07963=1204.555,411.485,-82.996,-175.840,8.484,148.473
C07964=1204.551,411.733,-83.032,-175.839,8.486,148.474
C07965=1204.547,411.980,-83.067,-175.839,8.488,148.474
C07966=1204.543,412.228,-83.102,-175.838,8.490,148.475
C07967=1204.540,412.475,-83.137,-175.838,8.493,148.475
C07968=1204.535,412.722,-83.172,-175.838,8.495,148.476
C07969=1204.531,412.970,-83.207,-175.837,8.497,148.476
C07970=1204.527,413.217,-83.242,-175.837,8.499,148.477
C07971=1204.523,413.464,-83.278,-175.837,8.501,148.477
C07972=1204.519,413.713,-83.313,-175.837,8.504,148.478
C07973=1204.515,413.959,-83.348,-175.836,8.506,148.478
C07974=1204.511,414.207,-83.384,-175.836,8.508,148.479
C07975=1204.508,414.455,-83.418,-175.836,8.510,148.479
C07976=1204.503,414.702,-83.454,-175.835,8.512,148.480
C07977=1204.499,414.950,-83.490,-175.835,8.514,148.480
C07978=1204.495,415.197,-83.525,-175.834,8.517,148.480
C07979=1204.491,415.444,-83.560,-175.834,8.519,148.481
C07980=1204.487,415.692,-83.595,-175.834,8.520,148.481
C07981=1204.483,415.939,-83.631,-175.834,8.522,148.482
C07982=1204.479,416.229,-83.671,-175.833,8.525,148.482
C07983=1204.475,416.518,-83.713,-175.833,8.528,148.483
C07984=1204.474,416.809,-83.754,-175.833,8.530,148.483
C07985=1204.475,417.097,-83.794,-175.832,8.532,148.484
C07986=1204.054,417.098,-83.832,-175.836,8.543,148.488
C07987=1204.052,416.805,-83.792,-175.836,8.541,148.487
C07988=1204.053,416.513,-83.750,-175.836,8.538,148.487
C07989=1204.057,416.220,-83.708,-175.836,8.536,148.486
C07990=1204.062,415.929,-83.667,-175.837,8.533,148.486
C07991=1204.065,415.681,-83.632,-175.837,8.531,148.485
C07992=1204.069,415.434,-83.596,-175.837,8.529,148.485
C07993=1204.074,415.187,-83.560,-175.838,8.527,148.484
C07994=1204.078,414.938,-83.526,-175.838,8.525,148.484
C07995=1204.082,414.691,-83.490,-175.838,8.523,148.483
C07996=1204.086,414.444,-83.455,-175.839,8.521,148.483
C07997=1204.090,414.196,-83.420,-175.839,8.518,148.482
C07998=1204.093,413.949,-83.384,-175.839,8.516,148.482
C07999=1204.098,413.702,-83.349,-175.839,8.514,148.481
C08000=1204.102,413.454,-83.314,-175.840,8.512,148.481
C08001=1204.105,413.206,-83.279,-175.840,8.510,148.480
C08002=1204.110,412.959,-83.244,-175.841,8.507,148.480
C08003=1204.114,412.711,-83.209,-175.841,8.505,148.479
C08004=1204.117,412.464,-83.173,-175.841,8.503,148.479
C08005=1204.121,412.217,-83.138,-175.842,8.501,148.478
C08006=1204.125,411.969,-83.103,-175.842,8.499,148.478
C08007=1204.129,411.721,-83.068,-175.842,8.496,148.477
C08008=1204.133,411.475,-83.033,-175.843,8.494,148.477
C08009=1204.137,411.226,-82.998,-175.843,8.492,148.476
C08010=1204.141,410.979,-82.962,-175.843,8.491,148.476
C08011=1204.145,410.732,-82.927,-175.843,8.488,148.475
C08012=1204.149,410.484,-82.892,-175.844,8.486,148.475
C08013=1204.153,410.237,-82.857,-175.844,8.483,148.475
C08014=1204.157,409.990,-82.821,-175.845,8.481,148.474
C08015=1204.161,409.742,-82.787,-175.845,8.479,148.474
C08016=1204.165,409.495,-82.751,-175.845,8.477,148.473
C08017=1204.169,409.247,-82.717,-175.846,8.475,148.473
C08018=1204.173,408.999,-82.681,-175.846,8.472,148.472
C08019=1204.177,408.752,-82.646,-175.846,8.470,148.472
C08020=1204.181,408.504,-82.611,-175.846,8.468,148.471
C08021=1204.185,408.257,-82.575,-175.847,8.466,148.471
C08022=1204.189,408.009,-82.541,-175.847,8.464,148.470
C08023=1204.193,407.762,-82.505,-175.847,8.461,148.470
C08024=1204.197,407.515,-82.470,-175.848,8.459,148.469
C08025=1204.201,407.267,-82.435,-175.848,8.457,148.469
C08026=1204.205,407.019,-82.400,-175.848,8.454,148.468
C08027=1204.210,406.772,-82.365,-175.849,8.453,148.468
C08028=1204.213,406.524,-82.330,-175.849,8.450,148.467
C08029=1204.218,406.277,-82.295,-175.849,8.448,148.467
C08030=1204.221,406.030,-82.260,-175.850,8.445,148.466
C08031=1204.225,405.781,-82.225,-175.850,8.443,148.466
C08032=1204.230,405.535,-82.190,-175.851,8.441,148.465
C08033=1204.234,405.286,-82.155,-175.851,8.438,148.465
C08034=1204.237,405.039,-82.119,-175.851,8.436,148.464
C08035=1204.242,404.792,-82.084,-175.852,8.434,148.464
C08036=1204.246,404.544,-82.049,-175.852,8.432,148.463
C08037=1204.250,404.297,-82.014,-175.852,8.430,148.463
C08038=1204.254,404.049,-81.979,-175.853,8.426,148.462
C08039=1204.258,403.802,-81.944,-175.853,8.424,148.462
C08040=1204.262,403.554,-81.909,-175.854,8.422,148.461
C08041=1204.265,403.306,-81.875,-175.854,8.420,148.461
C08042=1204.270,403.060,-81.840,-175.854,8.417,148.460
C08043=1204.274,402.811,-81.805,-175.855,8.415,148.460
C08044=1204.278,402.565,-81.770,-175.856,8.412,148.459
C08045=1204.282,402.317,-81.735,-175.856,8.410,148.459
C08046=1204.285,402.069,-81.700,-175.856,8.408,148.458
C08047=1204.290,401.822,-81.665,-175.856,8.406,148.457
C08048=1204.294,401.574,-81.630,-175.857,8.403,148.457
C08049=1204.298,401.327,-81.595,-175.858,8.400,148.457
C08050=1204.302,401.079,-81.560,-175.858,8.398,148.456
C08051=1204.306,400.832,-81.525,-175.858,8.396,148.456
C08052=1204.310,400.584,-81.491,-175.859,8.393,148.455
C08053=1204.313,400.337,-81.455,-175.859,8.391,148.454
C08054=1204.318,400.089,-81.421,-175.860,8.389,148.454
C08055=1204.322,399.842,-81.385,-175.861,8.385,148.453
C08056=1204.326,399.594,-81.351,-175.861,8.383,148.453
C08057=1204.330,399.346,-81.316,-175.861,8.381,148.452
C08058=1204.334,399.099,-81.281,-175.861,8.379,148.452
C08059=1204.338,398.851,-81.246,-175.862,8.376,148.451
C08060=1204.342,398.604,-81.212,-175.863,8.374,148.451
C08061=1204.346,398.357,-81.177,-175.863,8.371,148.450
C08062=1204.350,398.109,-81.142,-175.864,8.368,148.450
C08063=1204.354,397.862,-81.107,-175.864,8.366,148.449
C08064=1204.358,397.613,-81.072,-175.864,8.364,148.449
C08065=1204.363,397.366,-81.037,-175.865,8.361,148.448
C08066=1204.366,397.119,-81.002,-175.865,8.359,148.448
C08067=1204.370,396.871,-80.968,-175.866,8.355,148.447
C08068=1204.374,396.623,-80.933,-175.866,8.353,148.447
C08069=1204.379,396.376,-80.899,-175.867,8.351,148.446
C08070=1204.382,396.128,-80.863,-175.868,8.348,148.446
C08071=1204.387,395.881,-80.829,-175.868,8.346,148.445
C08072=1204.390,395.633,-80.794,-175.869,8.343,148.445
C08073=1204.394,395.386,-80.759,-175.869,8.341,148.444
C08074=1204.398,395.138,-80.724,-175.870,8.338,148.444
C08075=1204.403,394.891,-80.690,-175.871,8.335,148.443
C08076=1204.407,394.643,-80.655,-175.871,8.333,148.443
C08077=1204.410,394.396,-80.620,-175.872,8.330,148.442
C08078=1204.414,394.148,-80.586,-175.872,8.328,148.442
C08079=1204.419,393.901,-80.551,-175.873,8.325,148.441
C08080=1204.423,393.653,-80.516,-175.873,8.323,148.441
C08081=1204.426,393.406,-80.482,-175.874,8.320,148.440
C08082=1204.430,393.158,-80.447,-175.874,8.317,148.439
C08083=1204.435,392.875,-80.408,-175.875,8.314,148.439
C08084=1204.439,392.593,-80.368,-175.876,8.311,148.438
C08085=1204.444,392.310,-80.328,-175.876,8.308,148.438
C08086=1204.449,392.028,-80.289,-175.878,8.305,148.437
C08087=1204.453,391.780,-80.254,-175.878,8.302,148.437
C08088=1204.457,391.532,-80.220,-175.879,8.300,148.436
C08089=1204.461,391.285,-80.185,-175.879,8.297,148.436
C08090=1204.466,391.038,-80.150,-175.880,8.295,148.435
C08091=1204.469,390.790,-80.116,-175.881,8.292,148.435
C08092=1204.473,390.542,-80.081,-175.882,8.289,148.434
C08093=1204.477,390.294,-80.047,-175.882,8.286,148.434
C08094=1204.482,390.047,-80.012,-175.883,8.283,148.433
C08095=1204.485,389.800,-79.977,-175.883,8.281,148.433
C08096=1204.489,389.552,-79.943,-175.884,8.278,148.432
C08097=1204.493,389.304,-79.908,-175.885,8.275,148.432
C08098=1204.497,389.057,-79.874,-175.885,8.273,148.431
C08099=1204.501,388.809,-79.839,-175.886,8.270,148.430
C08100=1204.506,388.561,-79.805,-175.887,8.267,148.430
C08101=1204.510,388.314,-79.771,-175.888,8.265,148.430
C08102=1204.513,388.066,-79.736,-175.888,8.262,148.429
C08103=1204.518,387.819,-79.701,-175.890,8.259,148.429
C08104=1204.521,387.571,-79.667,-175.890,8.256,148.428
C08105=1204.526,387.324,-79.633,-175.891,8.254,148.427
C08106=1204.530,387.076,-79.597,-175.892,8.251,148.427
C08107=1204.533,386.829,-79.563,-175.893,8.248,148.426
C08108=1204.538,386.581,-79.529,-175.894,8.245,148.426
C08109=1204.542,386.333,-79.494,-175.894,8.243,148.426
C08110=1204.546,386.086,-79.460,-175.895,8.239,148.425
C08111=1204.550,385.838,-79.425,-175.896,8.237,148.425
C08112=1204.554,385.591,-79.391,-175.897,8.234,148.424
C08113=1204.557,385.343,-79.357,-175.898,8.231,148.424
C08114=1204.562,385.095,-79.322,-175.898,8.228,148.423
C08115=1204.566,384.848,-79.288,-175.899,8.226,148.423
C08116=1204.570,384.600,-79.253,-175.900,8.223,148.422
C08117=1204.574,384.353,-79.219,-175.901,8.219,148.421
C08118=1204.578,384.105,-79.185,-175.902,8.217,148.421
C08119=1204.582,383.858,-79.150,-175.903,8.214,148.420
C08120=1204.586,383.610,-79.117,-175.904,8.212,148.420
C08121=1204.590,383.362,-79.082,-175.904,8.208,148.420
C08122=1204.595,383.114,-79.048,-175.906,8.206,148.419
C08123=1204.598,382.867,-79.014,-175.906,8.203,148.419
C08124=1204.603,382.619,-78.979,-175.908,8.200,148.418
C08125=1204.607,382.372,-78.945,-175.908,8.197,148.418
C08126=1204.611,382.124,-78.910,-175.910,8.194,148.417
C08127=1204.614,381.877,-78.877,-175.910,8.191,148.417
C08128=1204.619,381.629,-78.842,-175.912,8.188,148.416
C08129=1204.622,381.382,-78.808,-175.913,8.185,148.416
C08130=1204.627,381.134,-78.774,-175.914,8.182,148.415
C08131=1204.632,380.886,-78.740,-175.915,8.179,148.415
C08132=1204.635,380.638,-78.705,-175.915,8.176,148.414
C08133=1204.639,380.391,-78.671,-175.917,8.173,148.414
C08134=1204.643,380.144,-78.637,-175.917,8.170,148.413
C08135=1204.647,379.896,-78.602,-175.919,8.167,148.413
C08136=1204.651,379.648,-78.569,-175.920,8.165,148.412
C08137=1204.656,379.400,-78.535,-175.921,8.161,148.412
C08138=1204.659,379.153,-78.500,-175.922,8.159,148.411
C08139=1204.664,378.905,-78.466,-175.923,8.156,148.411
C08140=1204.668,378.658,-78.432,-175.924,8.153,148.410
C08141=1204.672,378.409,-78.398,-175.925,8.150,148.410
C08142=1204.676,378.162,-78.364,-175.926,8.147,148.410
C08143=1204.680,377.915,-78.330,-175.927,8.144,148.409
C08144=1204.683,377.667,-78.295,-175.928,8.141,148.409
C08145=1204.688,377.419,-78.262,-175.929,8.138,148.408
C08146=1204.692,377.172,-78.228,-175.931,8.136,148.408
C08147=1204.695,376.924,-78.193,-175.931,8.132,148.407
C08148=1204.700,376.676,-78.160,-175.933,8.130,148.407
C08149=1204.704,376.429,-78.126,-175.934,8.126,148.407
C08150=1204.708,376.181,-78.091,-175.936,8.123,148.406
C08151=1204.712,375.933,-78.058,-175.936,8.120,148.406
C08152=1204.716,375.686,-78.024,-175.938,8.117,148.405
C08153=1204.721,375.439,-77.990,-175.939,8.114,148.405
C08154=1204.724,375.190,-77.956,-175.940,8.112,148.404
C08155=1204.729,374.943,-77.922,-175.941,8.109,148.404
C08156=1204.733,374.696,-77.888,-175.943,8.105,148.403
C08157=1204.736,374.447,-77.854,-175.944,8.102,148.403
C08158=1204.741,374.200,-77.820,-175.945,8.099,148.403
C08159=1204.744,373.953,-77.786,-175.946,8.097,148.402
C08160=1204.749,373.705,-77.752,-175.947,8.094,148.402
C08161=1204.753,373.457,-77.718,-175.949,8.090,148.401
C08162=1204.757,373.209,-77.685,-175.950,8.087,148.401
C08163=1204.761,372.962,-77.650,-175.952,8.084,148.401
C08164=1204.765,372.714,-77.617,-175.952,8.081,148.400
C08165=1204.769,372.466,-77.583,-175.954,8.078,148.400
C08166=1204.774,372.218,-77.549,-175.955,8.075,148.399
C08167=1204.777,371.971,-77.515,-175.957,8.072,148.399
C08168=1204.781,371.724,-77.481,-175.958,8.069,148.398
C08169=1204.785,371.475,-77.447,-175.959,8.066,148.398
C08170=1204.789,371.228,-77.413,-175.961,8.063,148.398
C08171=1204.793,370.980,-77.380,-175.962,8.060,148.397
C08172=1204.798,370.733,-77.347,-175.963,8.057,148.397
C08173=1204.802,370.485,-77.313,-175.965,8.054,148.396
C08174=1204.806,370.237,-77.279,-175.966,8.051,148.396
C08175=1204.810,369.990,-77.245,-175.967,8.048,148.396
C08176=1204.814,369.742,-77.211,-175.969,8.044,148.395
C08177=1204.818,369.494,-77.178,-175.970,8.041,148.395
C08178=1204.822,369.247,-77.144,-175.971,8.039,148.394
C08179=1204.826,368.999,-77.110,-175.974,8.035,148.394
C08180=1204.830,368.751,-77.076,-175.975,8.033,148.394
C08181=1204.835,368.503,-77.043,-175.976,8.030,148.393
C08182=1204.838,368.256,-77.009,-175.978,8.026,148.393
C08183=1204.843,368.008,-76.976,-175.979,8.023,148.392
C08184=1204.847,367.760,-76.942,-175.980,8.020,148.392
C08185=1204.851,367.512,-76.908,-175.982,8.017,148.392
C08186=1204.855,367.265,-76.875,-175.984,8.014,148.391
C08187=1204.860,366.984,-76.837,-175.985,8.011,148.391
C08188=1204.864,366.704,-76.799,-175.987,8.007,148.391
C08189=1204.869,366.423,-76.761,-175.989,8.003,148.390
C08190=1204.873,366.143,-76.723,-175.991,8.000,148.390
C08191=1204.877,365.895,-76.690,-175.992,7.997,148.389
C08192=1204.882,365.648,-76.656,-175.993,7.994,148.389
C08193=1204.885,365.399,-76.622,-175.995,7.991,148.389
C08194=1204.890,365.152,-76.589,-175.997,7.988,148.388
C08195=1204.894,364.904,-76.556,-175.998,7.984,148.388
C08196=1204.898,364.657,-76.522,-176.000,7.982,148.387
C08197=1204.902,364.409,-76.489,-176.002,7.978,148.387
C08198=1204.906,364.161,-76.456,-176.003,7.975,148.387
C08199=1204.910,363.914,-76.423,-176.004,7.973,148.386
C08200=1204.914,363.665,-76.388,-176.006,7.969,148.386
C08201=1204.918,363.418,-76.355,-176.008,7.966,148.386
C08202=1204.922,363.170,-76.321,-176.009,7.963,148.385
C08203=1204.926,362.922,-76.288,-176.011,7.960,148.385
C08204=1204.930,362.675,-76.255,-176.013,7.957,148.385
C08205=1204.935,362.427,-76.222,-176.015,7.954,148.385
C08206=1204.939,362.179,-76.189,-176.016,7.950,148.384
C08207=1204.943,361.931,-76.156,-176.017,7.948,148.384
C08208=1204.947,361.684,-76.122,-176.020,7.944,148.384
C08209=1204.951,361.437,-76.089,-176.021,7.941,148.383
C08210=1204.955,361.189,-76.055,-176.023,7.938,148.383
C08211=1204.959,360.940,-76.022,-176.024,7.935,148.383
C08212=1204.963,360.693,-75.989,-176.027,7.932,148.382
C08213=1204.967,360.445,-75.956,-176.028,7.929,148.382
C08214=1204.971,360.197,-75.922,-176.030,7.926,148.382
C08215=1204.975,359.950,-75.889,-176.031,7.923,148.381
C08216=1204.979,359.702,-75.856,-176.033,7.920,148.381
C08217=1204.983,359.454,-75.823,-176.035,7.917,148.381
C08218=1204.988,359.206,-75.790,-176.037,7.914,148.380
C08219=1204.992,358.959,-75.757,-176.039,7.910,148.380
C08220=1204.996,358.711,-75.724,-176.040,7.907,148.380
C08221=1205.000,358.463,-75.690,-176.042,7.904,148.379
C08222=1205.004,358.215,-75.657,-176.044,7.901,148.379
C08223=1205.008,357.968,-75.624,-176.046,7.898,148.379
C08224=1205.012,357.720,-75.591,-176.047,7.895,148.379
C08225=1205.016,357.472,-75.558,-176.049,7.892,148.378
C08226=1205.021,357.224,-75.525,-176.050,7.889,148.378
C08227=1205.025,356.976,-75.492,-176.053,7.886,148.378
C08228=1205.029,356.728,-75.459,-176.055,7.882,148.377
C08229=1205.033,356.481,-75.426,-176.056,7.879,148.377
C08230=1205.037,356.233,-75.393,-176.058,7.876,148.377
C08231=1205.041,355.986,-75.360,-176.060,7.874,148.377
C08232=1205.045,355.738,-75.327,-176.062,7.870,148.376
C08233=1205.049,355.490,-75.294,-176.063,7.867,148.376
C08234=1205.054,355.242,-75.261,-176.066,7.864,148.376
C08235=1205.058,354.994,-75.228,-176.067,7.860,148.375
C08236=1205.062,354.746,-75.195,-176.069,7.858,148.375
C08237=1205.066,354.499,-75.162,-176.071,7.855,148.375
C08238=1205.070,354.250,-75.129,-176.072,7.852,148.375
C08239=1205.074,354.003,-75.097,-176.075,7.848,148.374
C08240=1205.078,353.755,-75.064,-176.076,7.846,148.374
C08241=1205.082,353.507,-75.031,-176.079,7.843,148.374
C08242=1205.087,353.259,-74.998,-176.080,7.839,148.374
C08243=1205.091,353.011,-74.965,-176.082,7.836,148.373
C08244=1205.094,352.764,-74.932,-176.084,7.833,148.373
C08245=1205.099,352.516,-74.900,-176.086,7.831,148.373
C08246=1205.103,352.268,-74.867,-176.088,7.827,148.373
C08247=1205.107,352.021,-74.834,-176.090,7.824,148.372
C08248=1205.112,351.772,-74.802,-176.092,7.821,148.372
C08249=1205.115,351.525,-74.769,-176.094,7.818,148.372
C08250=1205.119,351.277,-74.736,-176.095,7.815,148.372
C08251=1205.124,351.029,-74.703,-176.098,7.812,148.371
C08252=1205.128,350.781,-74.670,-176.100,7.809,148.371
C08253=1205.131,350.534,-74.638,-176.101,7.806,148.371
C08254=1205.136,350.285,-74.605,-176.103,7.802,148.371
C08255=1205.141,350.038,-74.573,-176.105,7.800,148.370
C08256=1205.145,349.790,-74.540,-176.107,7.797,148.370
C08257=1205.148,349.543,-74.508,-176.109,7.793,148.370
C08258=1205.153,349.294,-74.475,-176.111,7.791,148.370
C08259=1205.157,349.046,-74.442,-176.113,7.787,148.370
C08260=1205.161,348.798,-74.410,-176.115,7.785,148.369
C08261=1205.165,348.551,-74.377,-176.117,7.781,148.369
C08262=1205.169,348.302,-74.344,-176.119,7.778,148.369
C08263=1205.173,348.056,-74.312,-176.121,7.775,148.369
C08264=1205.178,347.807,-74.280,-176.123,7.772,148.368
C08265=1205.182,347.560,-74.247,-176.124,7.769,148.368
C08266=1205.186,347.312,-74.215,-176.127,7.766,148.368
C08267=1205.190,347.064,-74.182,-176.129,7.763,148.368
C08268=1205.195,346.816,-74.150,-176.130,7.760,148.368
C08269=1205.198,346.569,-74.117,-176.133,7.757,148.367
C08270=1205.203,346.320,-74.085,-176.134,7.754,148.367
C08271=1205.207,346.072,-74.052,-176.137,7.751,148.367
C08272=1205.210,345.825,-74.020,-176.139,7.748,148.367
C08273=1205.215,345.576,-73.987,-176.140,7.745,148.367
C08274=1205.219,345.329,-73.956,-176.143,7.742,148.366
C08275=1205.223,345.081,-73.923,-176.144,7.739,148.366
C08276=1205.228,344.833,-73.890,-176.147,7.736,148.366
C08277=1205.232,344.585,-73.858,-176.149,7.733,148.366
C08278=1205.236,344.338,-73.825,-176.151,7.731,148.366
C08279=1205.240,344.090,-73.794,-176.153,7.727,148.365
C08280=1205.244,343.841,-73.761,-176.155,7.724,148.365
C08281=1205.248,343.593,-73.729,-176.157,7.721,148.365
C08282=1205.252,343.346,-73.696,-176.159,7.718,148.365
C08283=1205.257,343.098,-73.665,-176.161,7.715,148.365
C08284=1205.261,342.850,-73.632,-176.163,7.712,148.364
C08285=1205.265,342.602,-73.600,-176.165,7.709,148.364
C08286=1205.269,342.355,-73.568,-176.167,7.706,148.364
C08287=1205.273,342.107,-73.536,-176.169,7.703,148.364
C08288=1205.278,341.858,-73.503,-176.172,7.700,148.364
C08289=1205.281,341.610,-73.471,-176.173,7.697,148.364
C08290=1205.286,341.363,-73.439,-176.176,7.694,148.363
C08291=1205.291,341.084,-73.403,-176.178,7.691,148.363
C08292=1205.295,340.807,-73.367,-176.180,7.687,148.363
C08293=1205.300,340.528,-73.331,-176.182,7.684,148.363
C08294=1205.305,340.250,-73.295,-176.185,7.681,148.363
C08295=1205.309,340.002,-73.263,-176.187,7.678,148.363
C08296=1205.313,339.754,-73.230,-176.189,7.675,148.362
C08297=1205.317,339.507,-73.199,-176.191,7.672,148.362
C08298=1205.322,339.258,-73.166,-176.193,7.668,148.362
C08299=1205.325,339.010,-73.134,-176.195,7.666,148.362
C08300=1205.330,338.763,-73.103,-176.198,7.663,148.362
C08301=1205.334,338.515,-73.070,-176.199,7.660,148.362
C08302=1205.338,338.266,-73.039,-176.202,7.657,148.361
C08303=1205.342,338.019,-73.007,-176.204,7.654,148.361
C08304=1205.346,337.771,-72.975,-176.206,7.651,148.361
C08305=1205.350,337.523,-72.943,-176.208,7.648,148.361
C08306=1205.354,337.275,-72.911,-176.210,7.645,148.361
C08307=1205.359,337.027,-72.879,-176.212,7.643,148.361
C08308=1205.363,336.779,-72.847,-176.215,7.639,148.361
C08309=1205.367,336.532,-72.816,-176.217,7.636,148.360
C08310=1205.371,336.283,-72.783,-176.219,7.633,148.360
C08311=1205.375,336.035,-72.752,-176.221,7.630,148.360
C08312=1205.380,335.787,-72.721,-176.223,7.628,148.360
C08313=1205.384,335.539,-72.688,-176.225,7.625,148.360
C08314=1205.388,335.292,-72.657,-176.228,7.621,148.360
C08315=1205.392,335.044,-72.625,-176.229,7.619,148.360
C08316=1205.396,334.796,-72.593,-176.232,7.616,148.359
C08317=1205.401,334.548,-72.561,-176.234,7.613,148.359
C08318=1205.405,334.299,-72.530,-176.236,7.610,148.359
C08319=1205.409,334.051,-72.498,-176.238,7.607,148.359
C08320=1205.413,333.804,-72.466,-176.241,7.604,148.359
C08321=1205.417,333.556,-72.434,-176.243,7.601,148.359
C08322=1205.422,333.308,-72.403,-176.245,7.598,148.359
C08323=1205.426,333.060,-72.371,-176.247,7.596,148.359
C08324=1205.430,332.812,-72.340,-176.249,7.592,148.358
C08325=1205.434,332.564,-72.307,-176.252,7.589,148.358
C08326=1205.438,332.316,-72.276,-176.253,7.587,148.358
C08327=1205.443,332.068,-72.245,-176.256,7.583,148.358
C08328=1205.446,331.820,-72.213,-176.258,7.580,148.358
C08329=1205.451,331.572,-72.182,-176.260,7.578,148.358
C08330=1205.455,331.324,-72.150,-176.263,7.575,148.358
C08331=1205.460,331.076,-72.118,-176.265,7.572,148.358
C08332=1205.464,330.828,-72.086,-176.267,7.569,148.357
C08333=1205.468,330.580,-72.056,-176.269,7.566,148.357
C08334=1205.472,330.332,-72.024,-176.271,7.563,148.357
C08335=1205.476,330.085,-71.992,-176.274,7.560,148.357
C08336=1205.480,329.836,-71.961,-176.276,7.557,148.357
C08337=1205.484,329.589,-71.930,-176.278,7.555,148.357
C08338=1205.488,329.341,-71.898,-176.280,7.552,148.357
C08339=1205.494,329.093,-71.867,-176.283,7.549,148.357
C08340=1205.497,328.844,-71.835,-176.284,7.546,148.357
C08341=1205.502,328.597,-71.804,-176.287,7.543,148.357
C08342=1205.506,328.348,-71.772,-176.289,7.540,148.356
C08343=1205.510,328.101,-71.741,-176.291,7.537,148.356
C08344=1205.514,327.852,-71.710,-176.294,7.534,148.356
C08345=1205.518,327.605,-71.679,-176.296,7.532,148.356
C08346=1205.522,327.356,-71.647,-176.298,7.529,148.356
C08347=1205.527,327.109,-71.616,-176.301,7.526,148.356
C08348=1205.531,326.860,-71.584,-176.302,7.523,148.356
C08349=1205.535,326.613,-71.554,-176.305,7.520,148.356
C08350=1205.539,326.364,-71.522,-176.307,7.517,148.356
C08351=1205.543,326.117,-71.491,-176.309,7.514,148.356
C08352=1205.547,325.868,-71.460,-176.312,7.511,148.356
C08353=1205.552,325.621,-71.428,-176.314,7.508,148.356
C08354=1205.556,325.372,-71.397,-176.316,7.506,148.355
C08355=1205.560,325.125,-71.366,-176.319,7.503,148.355
C08356=1205.565,324.877,-71.335,-176.321,7.500,148.355
C08357=1205.569,324.628,-71.304,-176.323,7.497,148.355
C08358=1205.573,324.381,-71.272,-176.326,7.494,148.355
C08359=1205.577,324.132,-71.241,-176.327,7.491,148.355
C08360=1205.582,323.884,-71.210,-176.330,7.488,148.355
C08361=1205.585,323.636,-71.179,-176.333,7.485,148.355
C08362=1205.589,323.388,-71.148,-176.334,7.483,148.355
C08363=1205.594,323.140,-71.118,-176.337,7.480,148.355
C08364=1205.598,322.892,-71.086,-176.339,7.476,148.355
C08365=1205.602,322.644,-71.055,-176.341,7.474,148.355
C08366=1205.606,322.396,-71.024,-176.344,7.471,148.355
C08367=1205.611,322.148,-70.993,-176.346,7.469,148.355
C08368=1205.615,321.900,-70.962,-176.348,7.466,148.355
C08369=1205.619,321.652,-70.931,-176.351,7.462,148.354
C08370=1205.623,321.404,-70.900,-176.353,7.460,148.354
C08371=1205.628,321.156,-70.870,-176.355,7.457,148.354
C08372=1205.632,320.907,-70.839,-176.358,7.454,148.354
C08373=1205.636,320.659,-70.808,-176.360,7.452,148.354
C08374=1205.641,320.412,-70.776,-176.362,7.449,148.354
C08375=1205.645,320.163,-70.745,-176.365,7.445,148.354
C08376=1205.648,319.916,-70.715,-176.367,7.443,148.354
C08377=1205.653,319.668,-70.684,-176.369,7.440,148.354
C08378=1205.657,319.419,-70.653,-176.371,7.437,148.354
C08379=1205.662,319.171,-70.622,-176.374,7.434,148.354
C08380=1205.666,318.924,-70.592,-176.376,7.431,148.354
C08381=1205.670,318.675,-70.561,-176.379,7.429,148.354
C08382=1205.674,318.427,-70.530,-176.381,7.426,148.354
C08383=1205.679,318.179,-70.499,-176.383,7.423,148.354
C08384=1205.682,317.931,-70.469,-176.386,7.421,148.354
C08385=1205.686,317.683,-70.437,-176.388,7.417,148.354
C08386=1205.691,317.435,-70.407,-176.390,7.415,148.354
C08387=1205.695,317.186,-70.376,-176.393,7.412,148.354
C08388=1205.699,316.938,-70.346,-176.395,7.409,148.354
C08389=1205.704,316.691,-70.315,-176.397,7.407,148.353
C08390=1205.708,316.443,-70.285,-176.400,7.403,148.353
C08391=1205.712,316.194,-70.254,-176.402,7.400,148.353
C08392=1205.716,315.946,-70.223,-176.404,7.398,148.354
C08393=1205.721,315.698,-70.193,-176.407,7.395,148.353
C08394=1205.725,315.451,-70.162,-176.409,7.393,148.353
C08395=1205.729,315.174,-70.128,-176.411,7.390,148.353
C08396=1205.734,314.898,-70.094,-176.414,7.387,148.353
C08397=1205.739,314.622,-70.060,-176.417,7.384,148.353
C08398=1205.744,314.346,-70.026,-176.420,7.381,148.353
C08399=1205.748,314.098,-69.996,-176.422,7.377,148.353
C08400=1205.752,313.849,-69.965,-176.424,7.374,148.353
C08401=1205.756,313.601,-69.934,-176.427,7.372,148.353
C08402=1205.760,313.354,-69.904,-176.429,7.369,148.353
C08403=1205.765,313.106,-69.873,-176.432,7.366,148.353
C08404=1205.770,312.857,-69.843,-176.434,7.363,148.353
C08405=1205.773,312.609,-69.813,-176.436,7.360,148.353
C08406=1205.778,312.361,-69.782,-176.438,7.358,148.353
C08407=1205.782,312.113,-69.752,-176.441,7.355,148.353
C08408=1205.786,311.865,-69.722,-176.444,7.352,148.353
C08409=1205.790,311.617,-69.692,-176.445,7.350,148.353
C08410=1205.795,311.369,-69.661,-176.448,7.347,148.353
C08411=1205.799,311.120,-69.630,-176.450,7.344,148.353
C08412=1205.803,310.872,-69.600,-176.453,7.341,148.353
C08413=1205.808,310.624,-69.569,-176.456,7.338,148.353
C08414=1205.812,310.376,-69.540,-176.458,7.336,148.353
C08415=1205.817,310.128,-69.509,-176.460,7.333,148.353
C08416=1205.820,309.880,-69.479,-176.462,7.331,148.353
C08417=1205.825,309.631,-69.449,-176.465,7.328,148.353
C08418=1205.829,309.383,-69.418,-176.467,7.325,148.353
C08419=1205.833,309.135,-69.388,-176.470,7.322,148.353
C08420=1205.837,308.887,-69.358,-176.472,7.319,148.353
C08421=1205.841,308.639,-69.328,-176.474,7.317,148.353
C08422=1205.846,308.391,-69.298,-176.477,7.314,148.353
C08423=1205.850,308.143,-69.268,-176.480,7.311,148.353
C08424=1205.855,307.895,-69.238,-176.481,7.309,148.353
C08425=1205.859,307.647,-69.208,-176.484,7.306,148.353
C08426=1205.863,307.398,-69.177,-176.486,7.303,148.353
C08427=1205.867,307.150,-69.147,-176.489,7.300,148.353
C08428=1205.871,306.902,-69.118,-176.492,7.297,148.353
C08429=1205.876,306.654,-69.087,-176.494,7.295,148.353
C08430=1205.880,306.406,-69.057,-176.496,7.292,148.353
C08431=1205.885,306.158,-69.027,-176.499,7.290,148.353
C08432=1205.889,305.909,-68.997,-176.501,7.287,148.353
C08433=1205.893,305.662,-68.967,-176.504,7.284,148.353
C08434=1205.898,305.413,-68.937,-176.506,7.282,148.353
C08435=1205.902,305.165,-68.908,-176.509,7.279,148.353
C08436=1205.906,304.917,-68.877,-176.510,7.276,148.353
C08437=1205.911,304.669,-68.847,-176.513,7.273,148.353
C08438=1205.915,304.420,-68.818,-176.515,7.271,148.353
C08439=1205.919,304.173,-68.788,-176.518,7.268,148.353
C08440=1205.924,303.924,-68.758,-176.521,7.265,148.353
C08441=1205.928,303.676,-68.728,-176.523,7.263,148.353
C08442=1205.932,303.428,-68.698,-176.525,7.260,148.353
C08443=1205.936,303.180,-68.669,-176.527,7.257,148.353
C08444=1205.941,302.931,-68.639,-176.530,7.254,148.353
C08445=1205.945,302.684,-68.608,-176.533,7.251,148.353
C08446=1205.949,302.435,-68.579,-176.535,7.249,148.353
C08447=1205.954,302.187,-68.549,-176.538,7.246,148.353
C08448=1205.958,301.939,-68.519,-176.540,7.244,148.354
C08449=1205.962,301.691,-68.489,-176.542,7.241,148.354
C08450=1205.966,301.443,-68.460,-176.545,7.239,148.354
C08451=1205.970,301.194,-68.430,-176.547,7.236,148.354
C08452=1205.975,300.946,-68.400,-176.550,7.233,148.354
C08453=1205.979,300.698,-68.371,-176.552,7.230,148.354
C08454=1205.983,300.450,-68.341,-176.555,7.227,148.354
C08455=1205.987,300.202,-68.311,-176.557,7.225,148.354
C08456=1205.992,299.953,-68.282,-176.560,7.222,148.354
C08457=1205.996,299.705,-68.252,-176.562,7.220,148.354
C08458=1206.001,299.457,-68.222,-176.564,7.217,148.354
C08459=1206.005,299.208,-68.193,-176.567,7.215,148.354
C08460=1206.009,298.960,-68.163,-176.569,7.212,148.354
C08461=1206.013,298.712,-68.134,-176.572,7.209,148.354
C08462=1206.017,298.463,-68.104,-176.574,7.207,148.354
C08463=1206.021,298.216,-68.074,-176.577,7.204,148.354
C08464=1206.025,297.968,-68.045,-176.579,7.201,148.354
C08465=1206.030,297.719,-68.015,-176.582,7.199,148.354
C08466=1206.035,297.471,-67.986,-176.584,7.196,148.354
C08467=1206.039,297.223,-67.956,-176.587,7.193,148.354
C08468=1206.043,296.975,-67.927,-176.589,7.191,148.354
C08469=1206.048,296.727,-67.897,-176.592,7.188,148.355
C08470=1206.052,296.478,-67.868,-176.594,7.185,148.355
C08471=1206.056,296.230,-67.838,-176.597,7.183,148.355
C08472=1206.060,295.982,-67.809,-176.599,7.180,148.355
C08473=1206.065,295.733,-67.780,-176.601,7.178,148.355
C08474=1206.069,295.485,-67.751,-176.604,7.175,148.355
C08475=1206.074,295.237,-67.722,-176.606,7.173,148.355
C08476=1206.078,294.989,-67.692,-176.609,7.170,148.355
C08477=1206.082,294.741,-67.663,-176.611,7.167,148.355
C08478=1206.086,294.492,-67.633,-176.614,7.165,148.355
C08479=1206.090,294.244,-67.604,-176.616,7.162,148.355
C08480=1206.095,293.996,-67.574,-176.619,7.159,148.355
C08481=1206.099,293.747,-67.545,-176.621,7.157,148.355
C08482=1206.104,293.499,-67.517,-176.624,7.154,148.355
C08483=1206.108,293.251,-67.487,-176.626,7.151,148.355
C08484=1206.112,293.003,-67.458,-176.629,7.149,148.355
C08485=1206.116,292.754,-67.428,-176.631,7.146,148.355
C08486=1206.121,292.506,-67.399,-176.633,7.144,148.355
C08487=1206.126,292.258,-67.370,-176.637,7.141,148.356
C08488=1206.130,292.010,-67.341,-176.639,7.139,148.356
C08489=1206.133,291.762,-67.312,-176.641,7.136,148.356
C08490=1206.137,291.514,-67.283,-176.644,7.134,148.356
C08491=1206.142,291.265,-67.254,-176.646,7.131,148.356
C08492=1206.147,291.017,-67.225,-176.648,7.128,148.356
C08493=1206.151,290.769,-67.195,-176.651,7.125,148.356
C08494=1206.155,290.520,-67.167,-176.654,7.123,148.356
C08495=1206.160,290.272,-67.137,-176.656,7.120,148.356
C08496=1206.164,290.023,-67.108,-176.658,7.118,148.356
C08497=1206.169,289.775,-67.079,-176.661,7.115,148.356
C08498=1206.172,289.527,-67.050,-176.663,7.113,148.356
C08499=1206.178,289.253,-67.018,-176.666,7.110,148.356
C08500=1206.182,288.979,-66.986,-176.669,7.107,148.357
C08501=1206.187,288.704,-66.954,-176.672,7.104,148.357
C08502=1206.192,288.430,-66.923,-176.675,7.101,148.357
C08503=1206.196,288.182,-66.893,-176.677,7.099,148.357
C08504=1206.201,287.933,-66.864,-176.680,7.096,148.357
C08505=1206.204,287.685,-66.836,-176.682,7.094,148.357
C08506=1206.209,287.437,-66.807,-176.685,7.091,148.357
C08507=1206.213,287.189,-66.778,-176.687,7.089,148.357
C08508=1206.218,286.940,-66.749,-176.689,7.086,148.357
C08509=1206.222,286.692,-66.721,-176.692,7.084,148.357
C08510=1206.226,286.444,-66.692,-176.695,7.081,148.357
C08511=1206.230,286.195,-66.662,-176.697,7.079,148.358
C08512=1206.235,285.946,-66.634,-176.700,7.076,148.358
C08513=1206.239,285.699,-66.605,-176.702,7.074,148.358
C08514=1206.244,285.450,-66.576,-176.705,7.071,148.358
C08515=1206.248,285.201,-66.548,-176.707,7.069,148.358
C08516=1206.253,284.954,-66.519,-176.710,7.066,148.358
C08517=1206.257,284.705,-66.490,-176.712,7.064,148.358
C08518=1206.261,284.457,-66.461,-176.715,7.061,148.358
C08519=1206.266,284.209,-66.433,-176.717,7.059,148.358
C08520=1206.270,283.960,-66.404,-176.720,7.056,148.358
C08521=1206.274,283.713,-66.375,-176.722,7.053,148.358
C08522=1206.279,283.464,-66.347,-176.725,7.051,148.359
C08523=1206.283,283.215,-66.318,-176.727,7.049,148.359
C08524=1206.287,282.968,-66.289,-176.730,7.046,148.359
C08525=1206.292,282.719,-66.261,-176.732,7.043,148.359
C08526=1206.296,282.470,-66.232,-176.735,7.040,148.359
C08527=1206.300,282.223,-66.203,-176.737,7.038,148.359
C08528=1206.304,281.974,-66.175,-176.740,7.036,148.359
C08529=1206.309,281.726,-66.147,-176.742,7.033,148.359
C08530=1206.314,281.477,-66.118,-176.745,7.031,148.360
C08531=1206.317,281.229,-66.089,-176.748,7.028,148.360
C08532=1206.322,280.981,-66.061,-176.750,7.026,148.360
C08533=1206.326,280.732,-66.033,-176.752,7.023,148.360
C08534=1206.331,280.484,-66.004,-176.755,7.021,148.360
C08535=1206.335,280.235,-65.976,-176.758,7.018,148.360
C08536=1206.339,279.986,-65.948,-176.760,7.016,148.360
C08537=1206.343,279.739,-65.919,-176.762,7.013,148.360
C08538=1206.348,279.490,-65.890,-176.765,7.011,148.360
C08539=1206.352,279.242,-65.862,-176.767,7.009,148.361
C08540=1206.357,278.994,-65.834,-176.770,7.006,148.361
C08541=1206.361,278.746,-65.806,-176.773,7.004,148.361
C08542=1206.366,278.497,-65.777,-176.775,7.001,148.361
C08543=1206.370,278.249,-65.749,-176.777,6.999,148.361
C08544=1206.374,278.000,-65.721,-176.780,6.996,148.361
C08545=1206.378,277.751,-65.693,-176.783,6.994,148.361
C08546=1206.383,277.504,-65.663,-176.785,6.991,148.361
C08547=1206.387,277.255,-65.635,-176.788,6.989,148.361
C08548=1206.392,277.007,-65.607,-176.790,6.987,148.362
C08549=1206.395,276.759,-65.579,-176.793,6.984,148.362
C08550=1206.400,276.511,-65.551,-176.795,6.982,148.362
C08551=1206.404,276.262,-65.522,-176.798,6.979,148.362
C08552=1206.409,276.014,-65.495,-176.800,6.977,148.362
C08553=1206.413,275.764,-65.467,-176.803,6.974,148.362
C08554=1206.418,275.517,-65.439,-176.806,6.972,148.362
C08555=1206.422,275.268,-65.410,-176.808,6.970,148.363
C08556=1206.427,275.020,-65.382,-176.810,6.967,148.363
C08557=1206.430,274.771,-65.354,-176.813,6.965,148.363
C08558=1206.435,274.523,-65.326,-176.816,6.962,148.363
C08559=1206.439,274.274,-65.298,-176.818,6.960,148.363
C08560=1206.444,274.027,-65.270,-176.820,6.958,148.363
C08561=1206.449,273.778,-65.241,-176.823,6.955,148.363
C08562=1206.452,273.530,-65.213,-176.825,6.953,148.363
C08563=1206.457,273.281,-65.186,-176.828,6.950,148.364
C08564=1206.462,273.032,-65.157,-176.831,6.948,148.364
C08565=1206.466,272.785,-65.130,-176.833,6.945,148.364
C08566=1206.470,272.536,-65.102,-176.836,6.943,148.364
C08567=1206.475,272.288,-65.073,-176.838,6.941,148.364
C08568=1206.479,272.039,-65.046,-176.841,6.938,148.364
C08569=1206.483,271.791,-65.018,-176.843,6.936,148.364
C08570=1206.488,271.543,-64.990,-176.846,6.933,148.364
C08571=1206.492,271.294,-64.961,-176.848,6.931,148.365
C08572=1206.497,271.045,-64.934,-176.851,6.929,148.365
C08573=1206.500,270.797,-64.906,-176.853,6.926,148.365
C08574=1206.505,270.549,-64.878,-176.856,6.924,148.365
C08575=1206.510,270.301,-64.850,-176.859,6.921,148.365
C08576=1206.514,270.052,-64.823,-176.861,6.919,148.365
C08577=1206.518,269.804,-64.795,-176.864,6.917,148.366
C08578=1206.523,269.556,-64.767,-176.866,6.914,148.366
C08579=1206.527,269.306,-64.739,-176.868,6.912,148.366
C08580=1206.532,269.058,-64.711,-176.871,6.910,148.366
C08581=1206.536,268.810,-64.683,-176.874,6.907,148.366
C08582=1206.540,268.561,-64.656,-176.876,6.905,148.366
C08583=1206.545,268.314,-64.628,-176.879,6.902,148.366
C08584=1206.549,268.064,-64.601,-176.881,6.900,148.366
C08585=1206.554,267.816,-64.573,-176.884,6.898,148.367
C08586=1206.558,267.568,-64.546,-176.886,6.895,148.367
C08587=1206.562,267.319,-64.517,-176.889,6.893,148.367
C08588=1206.566,267.071,-64.490,-176.891,6.891,148.367
C08589=1206.571,266.823,-64.463,-176.894,6.888,148.367
C08590=1206.575,266.575,-64.435,-176.897,6.886,148.368
C08591=1206.579,266.326,-64.407,-176.899,6.883,148.368
C08592=1206.585,266.077,-64.379,-176.902,6.881,148.368
C08593=1206.589,265.829,-64.352,-176.904,6.879,148.368
C08594=1206.593,265.580,-64.324,-176.907,6.876,148.368
C08595=1206.598,265.332,-64.297,-176.909,6.874,148.368
C08596=1206.602,265.083,-64.270,-176.911,6.872,148.368
C08597=1206.606,264.835,-64.241,-176.915,6.869,148.369
C08598=1206.611,264.586,-64.214,-176.917,6.867,148.369
C08599=1206.615,264.338,-64.187,-176.919,6.865,148.369
C08600=1206.620,264.090,-64.160,-176.922,6.862,148.369
C08601=1206.623,263.841,-64.131,-176.925,6.860,148.369
C08602=1206.628,263.593,-64.104,-176.927,6.858,148.369
C08603=1206.633,263.320,-64.074,-176.930,6.855,148.370
C08604=1206.638,263.048,-64.044,-176.933,6.852,148.370
C08605=1206.643,262.775,-64.014,-176.935,6.850,148.370
C08606=1206.647,262.502,-63.984,-176.938,6.847,148.370
C08607=1206.652,262.254,-63.957,-176.941,6.845,148.370
C08608=1206.656,262.005,-63.930,-176.943,6.842,148.370
C08609=1206.660,261.756,-63.902,-176.946,6.841,148.371
C08610=1206.665,261.508,-63.875,-176.948,6.838,148.371
C08611=1206.669,261.260,-63.848,-176.951,6.836,148.371
C08612=1206.674,261.011,-63.820,-176.953,6.833,148.371
C08613=1206.678,260.762,-63.793,-176.956,6.832,148.371
C08614=1206.683,260.514,-63.765,-176.959,6.829,148.371
C08615=1206.687,260.266,-63.738,-176.961,6.827,148.372
C08616=1206.692,260.017,-63.711,-176.964,6.825,148.372
C08617=1206.696,259.769,-63.684,-176.967,6.822,148.372
C08618=1206.701,259.521,-63.656,-176.969,6.820,148.372
C08619=1206.705,259.272,-63.629,-176.971,6.818,148.373
C08620=1206.710,259.023,-63.602,-176.974,6.815,148.373
C08621=1206.713,258.775,-63.575,-176.976,6.813,148.373
C08622=1206.718,258.526,-63.548,-176.979,6.811,148.373
C08623=1206.723,258.278,-63.521,-176.981,6.809,148.373
C08624=1206.727,258.029,-63.494,-176.984,6.806,148.373
C08625=1206.732,257.780,-63.467,-176.986,6.804,148.373
C08626=1206.736,257.532,-63.439,-176.989,6.802,148.374
C08627=1206.740,257.284,-63.413,-176.992,6.799,148.374
C08628=1206.744,257.036,-63.385,-176.994,6.797,148.374
C08629=1206.749,256.787,-63.358,-176.996,6.795,148.374
C08630=1206.754,256.539,-63.331,-177.000,6.792,148.374
C08631=1206.758,256.290,-63.304,-177.002,6.790,148.375
C08632=1206.762,256.041,-63.277,-177.004,6.788,148.375
C08633=1206.766,255.793,-63.250,-177.007,6.786,148.375
C08634=1206.771,255.544,-63.223,-177.010,6.783,148.375
C08635=1206.776,255.296,-63.196,-177.012,6.781,148.375
C08636=1206.780,255.047,-63.169,-177.014,6.779,148.376
C08637=1206.784,254.799,-63.143,-177.018,6.776,148.376
C08638=1206.789,254.551,-63.116,-177.020,6.774,148.376
C08639=1206.794,254.302,-63.089,-177.022,6.772,148.376
C08640=1206.798,254.054,-63.062,-177.025,6.770,148.376
C08641=1206.802,253.806,-63.035,-177.028,6.768,148.377
C08642=1206.807,253.556,-63.009,-177.030,6.765,148.377
C08643=1206.811,253.307,-62.981,-177.033,6.764,148.377
C08644=1206.815,253.059,-62.955,-177.035,6.760,148.377
C08645=1206.820,252.811,-62.928,-177.038,6.759,148.377
C08646=1206.824,252.562,-62.901,-177.040,6.756,148.377
C08647=1206.828,252.314,-62.874,-177.043,6.755,148.378
C08648=1206.833,252.065,-62.847,-177.046,6.752,148.378
C08649=1206.838,251.816,-62.821,-177.048,6.750,148.378
C08650=1206.842,251.568,-62.794,-177.051,6.748,148.378
C08651=1206.847,251.320,-62.767,-177.053,6.746,148.379
C08652=1206.851,251.071,-62.740,-177.056,6.743,148.379
C08653=1206.855,250.823,-62.714,-177.058,6.741,148.379
C08654=1206.860,250.574,-62.687,-177.061,6.739,148.379
C08655=1206.865,250.325,-62.660,-177.063,6.737,148.379
C08656=1206.869,250.077,-62.634,-177.066,6.734,148.380
C08657=1206.873,249.829,-62.607,-177.069,6.732,148.380
C08658=1206.878,249.580,-62.581,-177.071,6.730,148.380
C08659=1206.882,249.331,-62.554,-177.073,6.728,148.380
C08660=1206.886,249.083,-62.528,-177.076,6.725,148.380
C08661=1206.891,248.834,-62.501,-177.079,6.723,148.381
C08662=1206.896,248.585,-62.474,-177.081,6.721,148.381
C08663=1206.900,248.337,-62.448,-177.084,6.719,148.381
C08664=1206.905,248.088,-62.421,-177.087,6.717,148.381
C08665=1206.909,247.840,-62.395,-177.089,6.714,148.381
C08666=1206.913,247.591,-62.368,-177.091,6.713,148.382
C08667=1206.917,247.343,-62.342,-177.094,6.710,148.382
C08668=1206.922,247.094,-62.315,-177.097,6.708,148.382
C08669=1206.926,246.845,-62.289,-177.099,6.706,148.382
C08670=1206.931,246.597,-62.262,-177.102,6.704,148.382
C08671=1206.935,246.349,-62.236,-177.104,6.702,148.383
C08672=1206.940,246.100,-62.210,-177.106,6.700,148.383
C08673=1206.944,245.852,-62.183,-177.110,6.697,148.383
C08674=1206.949,245.603,-62.157,-177.112,6.695,148.383
C08675=1206.953,245.355,-62.130,-177.114,6.693,148.384
C08676=1206.958,245.106,-62.104,-177.117,6.691,148.384
C08677=1206.962,244.858,-62.078,-177.120,6.688,148.384
C08678=1206.967,244.608,-62.051,-177.122,6.686,148.384
C08679=1206.971,244.360,-62.025,-177.125,6.684,148.385
C08680=1206.975,244.111,-61.999,-177.127,6.682,148.385
C08681=1206.980,243.863,-61.972,-177.130,6.680,148.385
C08682=1206.984,243.614,-61.946,-177.132,6.677,148.385
C08683=1206.989,243.366,-61.920,-177.135,6.676,148.385
C08684=1206.994,243.117,-61.894,-177.138,6.674,148.386
C08685=1206.998,242.869,-61.868,-177.140,6.671,148.386
C08686=1207.002,242.620,-61.841,-177.142,6.670,148.386
C08687=1207.007,242.371,-61.815,-177.146,6.667,148.386
C08688=1207.012,242.122,-61.789,-177.148,6.665,148.386
C08689=1207.016,241.874,-61.762,-177.150,6.663,148.387
C08690=1207.020,241.626,-61.737,-177.153,6.661,148.387
C08691=1207.025,241.377,-61.710,-177.155,6.659,148.387
C08692=1207.029,241.129,-61.684,-177.158,6.656,148.387
C08693=1207.033,240.880,-61.659,-177.160,6.654,148.388
C08694=1207.038,240.631,-61.632,-177.163,6.652,148.388
C08695=1207.042,240.383,-61.606,-177.166,6.650,148.388
C08696=1207.047,240.134,-61.580,-177.168,6.648,148.388
C08697=1207.051,239.886,-61.555,-177.171,6.646,148.389
C08698=1207.056,239.637,-61.528,-177.174,6.644,148.389
C08699=1207.060,239.388,-61.502,-177.176,6.641,148.389
C08700=1207.065,239.140,-61.476,-177.178,6.640,148.389
C08701=1207.070,238.891,-61.450,-177.181,6.638,148.390
C08702=1207.074,238.642,-61.424,-177.183,6.636,148.390
C08703=1207.078,238.394,-61.398,-177.186,6.633,148.390
C08704=1207.082,238.145,-61.372,-177.189,6.631,148.390
C08705=1207.087,237.896,-61.346,-177.191,6.629,148.390
C08706=1207.092,237.648,-61.320,-177.194,6.627,148.391
C08707=1207.097,237.377,-61.292,-177.197,6.624,148.391
C08708=1207.101,237.105,-61.264,-177.200,6.623,148.391
C08709=1207.107,236.834,-61.236,-177.202,6.621,148.392
C08710=1207.111,236.562,-61.207,-177.205,6.618,148.392
C08711=1207.115,236.314,-61.181,-177.208,6.616,148.392
C08712=1207.121,236.065,-61.155,-177.210,6.614,148.392
C08713=1207.125,235.816,-61.130,-177.212,6.612,148.392
C08714=1207.129,235.568,-61.104,-177.216,6.609,148.393
C08715=1207.133,235.319,-61.078,-177.218,6.607,148.393
C08716=1207.138,235.071,-61.053,-177.220,6.605,148.393
C08717=1207.143,234.822,-61.027,-177.223,6.603,148.393
C08718=1207.147,234.573,-61.001,-177.226,6.601,148.394
C08719=1207.152,234.325,-60.975,-177.228,6.600,148.394
C08720=1207.157,234.076,-60.950,-177.230,6.597,148.394
C08721=1207.161,233.827,-60.924,-177.234,6.595,148.394
C08722=1207.165,233.578,-60.898,-177.236,6.593,148.395
C08723=1207.170,233.330,-60.873,-177.238,6.591,148.395
C08724=1207.174,233.081,-60.847,-177.241,6.589,148.395
C08725=1207.178,232.833,-60.821,-177.244,6.587,148.396
C08726=1207.183,232.584,-60.796,-177.246,6.585,148.396
C08727=1207.187,232.336,-60.770,-177.248,6.583,148.396
C08728=1207.192,232.087,-60.744,-177.252,6.580,148.396
C08729=1207.197,231.838,-60.718,-177.254,6.578,148.397
C08730=1207.201,231.590,-60.692,-177.256,6.576,148.397
C08731=1207.206,231.341,-60.667,-177.259,6.574,148.397
C08732=1207.211,231.092,-60.642,-177.262,6.573,148.397
C08733=1207.215,230.843,-60.616,-177.264,6.571,148.398
C08734=1207.219,230.595,-60.591,-177.267,6.569,148.398
C08735=1207.224,230.346,-60.565,-177.269,6.567,148.398
C08736=1207.228,230.098,-60.539,-177.272,6.564,148.398
C08737=1207.233,229.850,-60.514,-177.275,6.562,148.399
C08738=1207.238,229.600,-60.489,-177.277,6.560,148.399
C08739=1207.242,229.351,-60.463,-177.280,6.558,148.399
C08740=1207.247,229.103,-60.438,-177.282,6.556,148.399
C08741=1207.251,228.854,-60.412,-177.285,6.555,148.400
C08742=1207.255,228.605,-60.388,-177.287,6.552,148.400
C08743=1207.259,228.357,-60.362,-177.290,6.551,148.400
C08744=1207.264,228.108,-60.337,-177.293,6.548,148.400
C08745=1207.268,227.860,-60.311,-177.296,6.546,148.401
C08746=1207.273,227.611,-60.286,-177.298,6.544,148.401
C08747=1207.277,227.362,-60.260,-177.300,6.542,148.401
C08748=1207.282,227.114,-60.235,-177.303,6.540,148.402
C08749=1207.287,226.864,-60.210,-177.306,6.538,148.402
C08750=1207.291,226.616,-60.185,-177.308,6.536,148.402
C08751=1207.296,226.368,-60.159,-177.310,6.534,148.402
C08752=1207.301,226.119,-60.134,-177.313,6.532,148.403
C08753=1207.304,225.870,-60.109,-177.316,6.530,148.403
C08754=1207.309,225.622,-60.084,-177.318,6.528,148.403
C08755=1207.314,225.373,-60.059,-177.321,6.526,148.403
C08756=1207.318,225.124,-60.033,-177.324,6.524,148.404
C08757=1207.323,224.875,-60.008,-177.326,6.522,148.404
C08758=1207.327,224.627,-59.982,-177.329,6.520,148.404
C08759=1207.332,224.378,-59.957,-177.331,6.518,148.404
C08760=1207.336,224.129,-59.933,-177.334,6.516,148.405
C08761=1207.341,223.881,-59.907,-177.336,6.514,148.405
C08762=1207.345,223.632,-59.882,-177.339,6.513,148.405
C08763=1207.350,223.384,-59.857,-177.342,6.510,148.406
C08764=1207.355,223.134,-59.832,-177.344,6.508,148.406
C08765=1207.359,222.886,-59.807,-177.347,6.506,148.406
C08766=1207.363,222.637,-59.782,-177.350,6.504,148.407
C08767=1207.368,222.389,-59.757,-177.352,6.502,148.407
C08768=1207.372,222.139,-59.732,-177.355,6.500,148.407
C08769=1207.377,221.892,-59.707,-177.357,6.498,148.407
C08770=1207.381,221.642,-59.682,-177.360,6.496,148.408
C08771=1207.386,221.394,-59.657,-177.362,6.494,148.408
C08772=1207.390,221.145,-59.631,-177.365,6.493,148.408
C08773=1207.395,220.896,-59.607,-177.368,6.491,148.409
C08774=1207.399,220.648,-59.581,-177.370,6.489,148.409
C08775=1207.404,220.399,-59.557,-177.373,6.486,148.409
C08776=1207.409,220.150,-59.533,-177.376,6.484,148.409
C08777=1207.413,219.902,-59.507,-177.378,6.482,148.410
C08778=1207.418,219.653,-59.482,-177.381,6.480,148.410
C08779=1207.422,219.404,-59.458,-177.384,6.479,148.410
C08780=1207.427,219.156,-59.432,-177.386,6.476,148.410
C08781=1207.431,218.906,-59.407,-177.388,6.475,148.411
C08782=1207.436,218.658,-59.383,-177.391,6.473,148.411
C08783=1207.440,218.410,-59.358,-177.394,6.471,148.411
C08784=1207.445,218.160,-59.333,-177.396,6.469,148.412
C08785=1207.449,217.912,-59.309,-177.399,6.467,148.412
C08786=1207.454,217.662,-59.284,-177.401,6.465,148.412
C08787=1207.459,217.414,-59.258,-177.404,6.463,148.413
C08788=1207.463,217.166,-59.234,-177.406,6.461,148.413
C08789=1207.468,216.917,-59.209,-177.409,6.460,148.413
C08790=1207.472,216.668,-59.185,-177.412,6.457,148.413
C08791=1207.476,216.419,-59.159,-177.415,6.455,148.414
C08792=1207.481,216.171,-59.135,-177.418,6.453,148.414
C08793=1207.486,215.922,-59.111,-177.420,6.451,148.414
C08794=1207.490,215.673,-59.086,-177.422,6.449,148.415
C08795=1207.495,215.424,-59.062,-177.425,6.447,148.415
C08796=1207.500,215.176,-59.037,-177.428,6.446,148.415
C08797=1207.503,214.927,-59.012,-177.430,6.444,148.416
C08798=1207.508,214.678,-58.987,-177.433,6.442,148.416
C08799=1207.512,214.429,-58.963,-177.436,6.440,148.416
C08800=1207.517,214.181,-58.938,-177.438,6.438,148.417
C08801=1207.522,213.932,-58.914,-177.440,6.436,148.417
C08802=1207.526,213.683,-58.889,-177.443,6.434,148.417
C08803=1207.531,213.434,-58.865,-177.446,6.432,148.417
C08804=1207.536,213.186,-58.840,-177.448,6.431,148.418
C08805=1207.540,212.937,-58.816,-177.451,6.429,148.418
C08806=1207.545,212.688,-58.791,-177.454,6.427,148.418
C08807=1207.549,212.439,-58.767,-177.456,6.425,148.419
C08808=1207.554,212.191,-58.742,-177.459,6.423,148.419
C08809=1207.558,211.941,-58.718,-177.461,6.421,148.419
C08810=1207.563,211.693,-58.693,-177.464,6.419,148.420
C08811=1207.568,211.423,-58.667,-177.467,6.417,148.420
C08812=1207.573,211.153,-58.640,-177.469,6.415,148.420
C08813=1207.577,210.882,-58.613,-177.473,6.413,148.421
C08814=1207.583,210.611,-58.587,-177.476,6.411,148.421
C08815=1207.587,210.363,-58.563,-177.478,6.408,148.421
C08816=1207.592,210.114,-58.539,-177.481,6.407,148.421
C08817=1207.596,209.865,-58.514,-177.483,6.405,148.422
C08818=1207.600,209.616,-58.490,-177.486,6.403,148.422
C08819=1207.606,209.368,-58.465,-177.489,6.401,148.422
C08820=1207.610,209.119,-58.441,-177.491,6.399,148.423
C08821=1207.614,208.870,-58.416,-177.494,6.397,148.423
C08822=1207.619,208.621,-58.393,-177.496,6.396,148.423
C08823=1207.624,208.372,-58.369,-177.499,6.394,148.424
C08824=1207.629,208.124,-58.344,-177.502,6.392,148.424
C08825=1207.632,207.875,-58.320,-177.504,6.390,148.424
C08826=1207.637,207.626,-58.296,-177.507,6.388,148.425
C08827=1207.642,207.377,-58.271,-177.509,6.386,148.425
C08828=1207.647,207.128,-58.248,-177.512,6.384,148.425
C08829=1207.651,206.880,-58.224,-177.515,6.382,148.426
C08830=1207.656,206.631,-58.199,-177.517,6.381,148.426
C08831=1207.660,206.382,-58.174,-177.520,6.379,148.426
C08832=1207.665,206.133,-58.151,-177.522,6.377,148.427
C08833=1207.669,205.885,-58.127,-177.525,6.375,148.427
C08834=1207.674,205.636,-58.102,-177.528,6.373,148.427
C08835=1207.679,205.388,-58.078,-177.530,6.371,148.428
C08836=1207.683,205.138,-58.055,-177.533,6.370,148.428
C08837=1207.687,204.889,-58.030,-177.536,6.368,148.428
C08838=1207.692,204.641,-58.006,-177.538,6.366,148.429
C08839=1207.697,204.392,-57.982,-177.541,6.364,148.429
C08840=1207.701,204.143,-57.958,-177.543,6.362,148.429
C08841=1207.706,203.895,-57.934,-177.546,6.360,148.429
C08842=1207.710,203.645,-57.911,-177.548,6.358,148.430
C08843=1207.715,203.396,-57.886,-177.551,6.356,148.430
C08844=1207.720,203.147,-57.863,-177.554,6.355,148.430
C08845=1207.724,202.899,-57.838,-177.556,6.353,148.431
C08846=1207.728,202.651,-57.814,-177.559,6.351,148.431
C08847=1207.733,202.401,-57.791,-177.561,6.350,148.432
C08848=1207.738,202.153,-57.766,-177.564,6.348,148.432
C08849=1207.743,201.904,-57.743,-177.566,6.346,148.432
C08850=1207.747,201.655,-57.719,-177.569,6.345,148.433
C08851=1207.752,201.406,-57.695,-177.572,6.343,148.433
C08852=1207.756,201.157,-57.671,-177.574,6.341,148.433
C08853=1207.761,200.908,-57.648,-177.577,6.339,148.434
C08854=1207.765,200.660,-57.624,-177.580,6.337,148.434
C08855=1207.770,200.411,-57.600,-177.582,6.335,148.434
C08856=1207.775,200.162,-57.576,-177.585,6.334,148.435
C08857=1207.780,199.913,-57.552,-177.588,6.332,148.435
C08858=1207.784,199.665,-57.528,-177.590,6.330,148.435
C08859=1207.789,199.415,-57.505,-177.593,6.328,148.436
C08860=1207.793,199.167,-57.481,-177.596,6.326,148.436
C08861=1207.797,198.917,-57.457,-177.598,6.324,148.436
C08862=1207.801,198.669,-57.433,-177.601,6.323,148.437
C08863=1207.806,198.420,-57.410,-177.603,6.321,148.437
C08864=1207.811,198.171,-57.386,-177.606,6.319,148.437
C08865=1207.815,197.922,-57.362,-177.609,6.317,148.438
C08866=1207.820,197.673,-57.339,-177.611,6.315,148.438
C08867=1207.825,197.424,-57.315,-177.613,6.314,148.438
C08868=1207.829,197.176,-57.291,-177.616,6.312,148.439
C08869=1207.834,196.927,-57.268,-177.618,6.310,148.439
C08870=1207.838,196.679,-57.244,-177.621,6.308,148.439
C08871=1207.843,196.430,-57.221,-177.624,6.307,148.440
C08872=1207.848,196.180,-57.197,-177.626,6.305,148.440
C08873=1207.852,195.931,-57.174,-177.629,6.303,148.440
C08874=1207.857,195.683,-57.150,-177.632,6.301,148.441
C08875=1207.861,195.434,-57.126,-177.634,6.299,148.441
C08876=1207.866,195.185,-57.103,-177.637,6.298,148.441
C08877=1207.871,194.936,-57.080,-177.640,6.296,148.442
C08878=1207.875,194.688,-57.056,-177.642,6.294,148.442
C08879=1207.880,194.438,-57.032,-177.645,6.292,148.442
C08880=1207.885,194.189,-57.009,-177.647,6.291,148.443
C08881=1207.889,193.940,-56.986,-177.650,6.289,148.443
C08882=1207.894,193.692,-56.962,-177.652,6.287,148.443
C08883=1207.898,193.443,-56.938,-177.655,6.286,148.444
C08884=1207.902,193.194,-56.915,-177.658,6.284,148.444
C08885=1207.907,192.945,-56.892,-177.661,6.282,148.445
C08886=1207.912,192.697,-56.869,-177.663,6.280,148.445
C08887=1207.917,192.448,-56.846,-177.666,6.279,148.445
C08888=1207.921,192.199,-56.822,-177.669,6.277,148.446
C08889=1207.926,191.950,-56.798,-177.671,6.275,148.446
C08890=1207.931,191.701,-56.775,-177.674,6.273,148.446
C08891=1207.936,191.452,-56.752,-177.676,6.272,148.447
C08892=1207.939,191.204,-56.729,-177.679,6.270,148.447
C08893=1207.944,190.955,-56.705,-177.681,6.269,148.448
C08894=1207.949,190.706,-56.682,-177.684,6.267,148.448
C08895=1207.954,190.457,-56.659,-177.687,6.265,148.448
C08896=1207.958,190.207,-56.635,-177.689,6.263,148.449
C08897=1207.964,189.959,-56.612,-177.692,6.261,148.449
C08898=1207.968,189.710,-56.590,-177.695,6.259,148.449
C08899=1207.972,189.461,-56.566,-177.697,6.258,148.450
C08900=1207.977,189.212,-56.543,-177.699,6.257,148.450
C08901=1207.982,188.963,-56.520,-177.702,6.255,148.450
C08902=1207.986,188.715,-56.497,-177.705,6.253,148.451
C08903=1207.990,188.466,-56.473,-177.707,6.251,148.451
C08904=1207.995,188.217,-56.450,-177.710,6.249,148.451
C08905=1208.000,187.968,-56.427,-177.713,6.248,148.452
C08906=1208.004,187.720,-56.404,-177.715,6.246,148.452
C08907=1208.009,187.470,-56.381,-177.717,6.245,148.453
C08908=1208.014,187.221,-56.358,-177.720,6.243,148.453
C08909=1208.018,186.972,-56.334,-177.723,6.241,148.453
C08910=1208.022,186.724,-56.311,-177.725,6.239,148.454
C08911=1208.027,186.475,-56.288,-177.728,6.237,148.454
C08912=1208.033,186.226,-56.266,-177.731,6.236,148.454
C08913=1208.037,185.977,-56.243,-177.734,6.234,148.455
C08914=1208.041,185.728,-56.220,-177.736,6.232,148.455
C08915=1208.047,185.458,-56.195,-177.739,6.231,148.456
C08916=1208.051,185.189,-56.170,-177.742,6.229,148.456
C08917=1208.057,184.919,-56.145,-177.744,6.227,148.456
C08918=1208.062,184.649,-56.120,-177.748,6.225,148.457
C08919=1208.066,184.400,-56.097,-177.750,6.224,148.457
C08920=1208.070,184.151,-56.074,-177.753,6.222,148.458
C08921=1208.076,183.903,-56.051,-177.755,6.221,148.458
C08922=1208.080,183.654,-56.028,-177.758,6.219,148.458
C08923=1208.085,183.405,-56.006,-177.760,6.217,148.459
C08924=1208.089,183.156,-55.983,-177.763,6.215,148.459
C08925=1208.093,182.907,-55.959,-177.766,6.214,148.459
C08926=1208.099,182.659,-55.936,-177.768,6.212,148.460
C08927=1208.103,182.409,-55.914,-177.770,6.211,148.460
C08928=1208.108,182.160,-55.891,-177.773,6.209,148.460
C08929=1208.112,181.912,-55.868,-177.776,6.207,148.461
C08930=1208.117,181.663,-55.846,-177.779,6.206,148.461
C08931=1208.121,181.414,-55.823,-177.781,6.204,148.462
C08932=1208.126,181.165,-55.800,-177.784,6.202,148.462
C08933=1208.130,180.916,-55.778,-177.786,6.201,148.462
C08934=1208.135,180.667,-55.755,-177.789,6.199,148.463
C08935=1208.140,180.418,-55.732,-177.792,6.197,148.463
C08936=1208.144,180.169,-55.709,-177.794,6.196,148.464
C08937=1208.150,179.920,-55.686,-177.797,6.194,148.464
C08938=1208.154,179.671,-55.664,-177.799,6.192,148.464
C08939=1208.159,179.422,-55.641,-177.802,6.191,148.465
C08940=1208.163,179.173,-55.618,-177.805,6.189,148.465
C08941=1208.168,178.924,-55.596,-177.807,6.188,148.466
C08942=1208.172,178.676,-55.573,-177.810,6.186,148.466
C08943=1208.177,178.426,-55.551,-177.813,6.184,148.466
C08944=1208.182,178.178,-55.528,-177.815,6.183,148.467
C08945=1208.186,177.929,-55.506,-177.817,6.181,148.467
C08946=1208.191,177.680,-55.483,-177.820,6.179,148.467
C08947=1208.196,177.431,-55.461,-177.823,6.178,148.468
C08948=1208.200,177.182,-55.438,-177.825,6.176,148.468
C08949=1208.205,176.933,-55.416,-177.828,6.175,148.469
C08950=1208.210,176.684,-55.393,-177.831,6.173,148.469
C08951=1208.214,176.435,-55.371,-177.833,6.171,148.469
C08952=1208.218,176.186,-55.348,-177.836,6.170,148.470
C08953=1208.224,175.937,-55.326,-177.839,6.168,148.470
C08954=1208.228,175.688,-55.304,-177.841,6.167,148.471
C08955=1208.233,175.439,-55.280,-177.843,6.165,148.471
C08956=1208.238,175.190,-55.259,-177.846,6.163,148.471
C08957=1208.242,174.942,-55.236,-177.849,6.162,148.472
C08958=1208.247,174.693,-55.214,-177.851,6.161,148.472
C08959=1208.251,174.443,-55.191,-177.854,6.159,148.473
C08960=1208.255,174.195,-55.169,-177.857,6.157,148.473
C08961=1208.261,173.946,-55.146,-177.859,6.155,148.473
C08962=1208.265,173.696,-55.124,-177.862,6.154,148.474
C08963=1208.270,173.448,-55.102,-177.864,6.153,148.474
C08964=1208.275,173.199,-55.079,-177.867,6.151,148.475
C08965=1208.279,172.949,-55.057,-177.870,6.149,148.475
C08966=1208.284,172.701,-55.035,-177.873,6.147,148.475
C08967=1208.289,172.452,-55.012,-177.875,6.146,148.476
C08968=1208.294,172.203,-54.991,-177.877,6.145,148.476
C08969=1208.298,171.954,-54.968,-177.880,6.143,148.476
C08970=1208.303,171.705,-54.946,-177.883,6.141,148.477
C08971=1208.307,171.456,-54.923,-177.886,6.140,148.477
C08972=1208.312,171.207,-54.901,-177.888,6.139,148.478
C08973=1208.317,170.958,-54.880,-177.891,6.137,148.478
C08974=1208.321,170.709,-54.856,-177.893,6.135,148.479
C08975=1208.326,170.460,-54.835,-177.896,6.133,148.479
C08976=1208.330,170.211,-54.813,-177.898,6.132,148.479
C08977=1208.335,169.962,-54.791,-177.901,6.131,148.480
C08978=1208.340,169.713,-54.768,-177.904,6.129,148.480
C08979=1208.345,169.465,-54.746,-177.906,6.127,148.481
C08980=1208.349,169.215,-54.724,-177.909,6.126,148.481
C08981=1208.354,168.967,-54.702,-177.911,6.124,148.481
C08982=1208.358,168.717,-54.680,-177.914,6.123,148.482
C08983=1208.364,168.468,-54.658,-177.917,6.121,148.482
C08984=1208.368,168.219,-54.636,-177.919,6.120,148.483
C08985=1208.373,167.970,-54.614,-177.922,6.118,148.483
C08986=1208.377,167.721,-54.592,-177.924,6.116,148.483
C08987=1208.382,167.473,-54.570,-177.927,6.115,148.484
C08988=1208.387,167.223,-54.547,-177.929,6.114,148.484
C08989=1208.392,166.975,-54.525,-177.932,6.112,148.485
C08990=1208.396,166.725,-54.503,-177.935,6.110,148.485
C08991=1208.401,166.477,-54.482,-177.937,6.109,148.485
C08992=1208.405,166.227,-54.460,-177.940,6.108,148.486
C08993=1208.410,165.979,-54.438,-177.942,6.106,148.486
C08994=1208.414,165.729,-54.416,-177.946,6.104,148.487
C08995=1208.419,165.481,-54.394,-177.948,6.103,148.487
C08996=1208.423,165.231,-54.372,-177.950,6.102,148.488
C08997=1208.429,164.982,-54.350,-177.953,6.100,148.488
C08998=1208.433,164.733,-54.328,-177.955,6.099,148.488
C08999=1208.438,164.485,-54.306,-177.958,6.097,148.489
C09000=1208.443,164.236,-54.284,-177.961,6.096,148.489
C09001=1208.447,163.987,-54.262,-177.964,6.094,148.490
C09002=1208.452,163.737,-54.241,-177.966,6.093,148.490
C09003=1208.457,163.488,-54.219,-177.968,6.091,148.490
C09004=1208.462,163.239,-54.198,-177.972,6.089,148.491
C09005=1208.466,162.990,-54.176,-177.974,6.088,148.491
C09006=1208.471,162.741,-54.154,-177.976,6.087,148.492
C09007=1208.476,162.493,-54.132,-177.979,6.085,148.492
C09008=1208.480,162.243,-54.110,-177.982,6.083,148.492
C09009=1208.485,161.995,-54.089,-177.984,6.082,148.493
C09010=1208.489,161.745,-54.066,-177.987,6.081,148.493
C09011=1208.494,161.496,-54.046,-177.990,6.079,148.494
C09012=1208.499,161.247,-54.024,-177.992,6.078,148.494
C09013=1208.503,160.998,-54.002,-177.995,6.076,148.495
C09014=1208.508,160.749,-53.980,-177.998,6.075,148.495
C09015=1208.513,160.501,-53.958,-178.000,6.074,148.496
C09016=1208.518,160.251,-53.937,-178.002,6.072,148.496
C09017=1208.522,160.002,-53.915,-178.005,6.070,148.496
C09018=1208.527,159.753,-53.893,-178.008,6.069,148.497
C09019=1208.531,159.484,-53.871,-178.010,6.068,148.497
C09020=1208.537,159.215,-53.847,-178.013,6.066,148.498
C09021=1208.542,158.947,-53.824,-178.016,6.064,148.498
C09022=1208.547,158.677,-53.801,-178.019,6.063,148.499
C09023=1208.552,158.428,-53.779,-178.022,6.061,148.499
C09024=1208.557,158.179,-53.757,-178.024,6.060,148.500
C09025=1208.562,157.930,-53.736,-178.027,6.058,148.500
C09026=1208.566,157.681,-53.714,-178.029,6.056,148.500
C09027=1208.570,157.432,-53.693,-178.032,6.056,148.501
C09028=1208.575,157.183,-53.672,-178.035,6.054,148.501
C09029=1208.580,156.934,-53.650,-178.037,6.052,148.502
C09030=1208.585,156.685,-53.629,-178.039,6.051,148.502
C09031=1208.590,156.436,-53.607,-178.043,6.050,148.503
C09032=1208.594,156.187,-53.585,-178.045,6.048,148.503
C09033=1208.599,155.937,-53.564,-178.047,6.047,148.503
C09034=1208.603,155.689,-53.543,-178.050,6.045,148.504
C09035=1208.608,155.440,-53.522,-178.053,6.044,148.504
C09036=1208.613,155.190,-53.500,-178.055,6.043,148.505
C09037=1208.618,154.942,-53.478,-178.058,6.041,148.505
C09038=1208.623,154.693,-53.458,-178.061,6.039,148.506
C09039=1208.627,154.443,-53.435,-178.063,6.039,148.506
C09040=1208.631,154.194,-53.415,-178.066,6.037,148.507
C09041=1208.636,153.946,-53.393,-178.069,6.035,148.507
C09042=1208.641,153.696,-53.372,-178.071,6.034,148.507
C09043=1208.646,153.448,-53.351,-178.074,6.033,148.508
C09044=1208.650,153.198,-53.330,-178.076,6.031,148.508
C09045=1208.655,152.949,-53.308,-178.079,6.030,148.509
C09046=1208.660,152.700,-53.287,-178.081,6.028,148.509
C09047=1208.665,152.452,-53.266,-178.084,6.027,148.510
C09048=1208.669,152.202,-53.245,-178.087,6.026,148.510
C09049=1208.674,151.953,-53.223,-178.089,6.024,148.510
C09050=1208.679,151.704,-53.202,-178.092,6.023,148.511
C09051=1208.684,151.455,-53.181,-178.094,6.021,148.511
C09052=1208.688,151.206,-53.160,-178.097,6.020,148.512
C09053=1208.693,150.956,-53.139,-178.099,6.019,148.512
C09054=1208.698,150.708,-53.117,-178.102,6.017,148.513
C09055=1208.702,150.459,-53.097,-178.105,6.015,148.513
C09056=1208.707,150.210,-53.076,-178.107,6.014,148.514
C09057=1208.712,149.961,-53.054,-178.110,6.013,148.514
C09058=1208.716,149.711,-53.033,-178.112,6.012,148.515
C09059=1208.721,149.462,-53.013,-178.115,6.010,148.515
C09060=1208.726,149.213,-52.991,-178.118,6.008,148.515
C09061=1208.731,148.964,-52.970,-178.120,6.008,148.516
C09062=1208.736,148.715,-52.949,-178.123,6.006,148.516
C09063=1208.741,148.467,-52.928,-178.126,6.004,148.517
C09064=1208.744,148.217,-52.907,-178.128,6.003,148.517
C09065=1208.750,147.968,-52.886,-178.131,6.002,148.518
C09066=1208.754,147.719,-52.864,-178.133,6.001,148.518
C09067=1208.759,147.470,-52.844,-178.136,5.999,148.519
C09068=1208.764,147.221,-52.823,-178.139,5.997,148.519
C09069=1208.768,146.972,-52.803,-178.141,5.997,148.520
C09070=1208.774,146.723,-52.782,-178.144,5.995,148.520
C09071=1208.778,146.473,-52.760,-178.146,5.994,148.521
C09072=1208.782,146.224,-52.739,-178.149,5.992,148.521
C09073=1208.788,145.975,-52.718,-178.152,5.991,148.521
C09074=1208.792,145.726,-52.698,-178.154,5.990,148.522
C09075=1208.797,145.477,-52.677,-178.157,5.988,148.522
C09076=1208.801,145.228,-52.656,-178.159,5.987,148.523
C09077=1208.806,144.979,-52.635,-178.162,5.986,148.523
C09078=1208.811,144.730,-52.615,-178.165,5.984,148.524
C09079=1208.816,144.481,-52.594,-178.167,5.983,148.524
C09080=1208.821,144.232,-52.573,-178.170,5.981,148.525
C09081=1208.825,143.982,-52.552,-178.172,5.981,148.525
C09082=1208.830,143.733,-52.532,-178.175,5.979,148.525
C09083=1208.834,143.485,-52.510,-178.178,5.978,148.526
C09084=1208.839,143.236,-52.489,-178.180,5.976,148.526
C09085=1208.844,142.986,-52.469,-178.183,5.975,148.527
C09086=1208.848,142.737,-52.448,-178.186,5.974,148.527
C09087=1208.854,142.488,-52.427,-178.188,5.972,148.528
C09088=1208.858,142.239,-52.407,-178.190,5.971,148.528
C09089=1208.863,141.990,-52.386,-178.193,5.970,148.529
C09090=1208.868,141.741,-52.365,-178.196,5.969,148.529
C09091=1208.873,141.492,-52.345,-178.198,5.967,148.530
C09092=1208.877,141.243,-52.324,-178.201,5.965,148.530
C09093=1208.882,140.994,-52.304,-178.204,5.965,148.531
C09094=1208.887,140.745,-52.283,-178.206,5.963,148.531
C09095=1208.891,140.496,-52.262,-178.209,5.962,148.532
C09096=1208.897,140.246,-52.241,-178.212,5.960,148.532
C09097=1208.901,139.997,-52.221,-178.214,5.959,148.532
C09098=1208.905,139.748,-52.201,-178.217,5.958,148.533
C09099=1208.911,139.499,-52.180,-178.219,5.956,148.533
C09100=1208.915,139.250,-52.159,-178.222,5.955,148.534
C09101=1208.920,139.001,-52.138,-178.225,5.954,148.534
C09102=1208.925,138.752,-52.118,-178.227,5.953,148.535
C09103=1208.929,138.502,-52.098,-178.230,5.951,148.535
C09104=1208.935,138.253,-52.077,-178.232,5.950,148.536
C09105=1208.939,138.004,-52.057,-178.235,5.949,148.536
C09106=1208.943,137.755,-52.037,-178.237,5.948,148.537
C09107=1208.949,137.506,-52.016,-178.240,5.946,148.537
C09108=1208.953,137.257,-51.995,-178.242,5.945,148.538
C09109=1208.957,137.008,-51.975,-178.245,5.944,148.538
C09110=1208.963,136.759,-51.954,-178.248,5.942,148.539
C09111=1208.967,136.509,-51.934,-178.250,5.941,148.539
C09112=1208.972,136.260,-51.914,-178.253,5.940,148.540
C09113=1208.977,136.011,-51.893,-178.255,5.939,148.540
C09114=1208.981,135.762,-51.873,-178.259,5.937,148.541
C09115=1208.986,135.513,-51.852,-178.261,5.936,148.541
C09116=1208.991,135.264,-51.833,-178.263,5.934,148.541
C09117=1208.996,135.014,-51.812,-178.266,5.934,148.542
C09118=1209.000,134.765,-51.791,-178.269,5.932,148.542
C09119=1209.005,134.517,-51.771,-178.271,5.931,148.543
C09120=1209.010,134.268,-51.752,-178.274,5.930,148.543
C09121=1209.015,134.018,-51.731,-178.276,5.929,148.544
C09122=1209.020,133.769,-51.710,-178.279,5.927,148.545
C09123=1209.025,133.501,-51.689,-178.282,5.925,148.545
C09124=1209.030,133.232,-51.667,-178.285,5.925,148.546
C09125=1209.035,132.963,-51.645,-178.287,5.923,148.546
C09126=1209.040,132.695,-51.623,-178.290,5.922,148.547
C09127=1209.044,132.445,-51.603,-178.293,5.921,148.547
C09128=1209.050,132.197,-51.583,-178.296,5.919,148.548
C09129=1209.054,131.948,-51.562,-178.298,5.918,148.548
C09130=1209.059,131.698,-51.543,-178.301,5.917,148.549
C09131=1209.064,131.449,-51.522,-178.303,5.916,148.549
C09132=1209.068,131.200,-51.503,-178.306,5.914,148.549
C09133=1209.074,130.950,-51.482,-178.308,5.913,148.550
